RoboDK station: kr10 0621 Cube.rdk

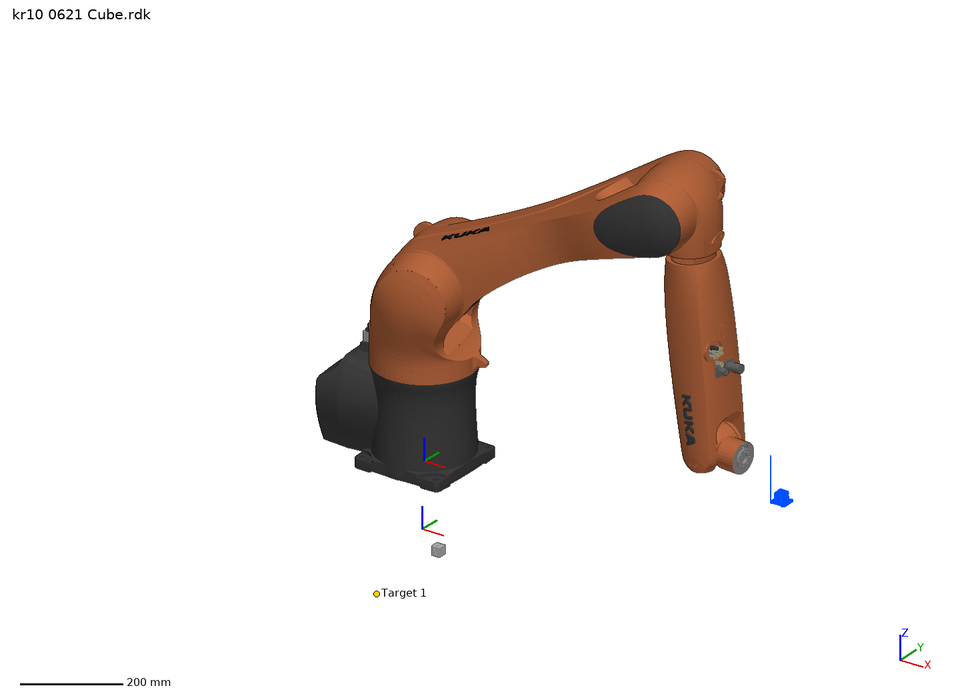
[picture v0: the station drawn from its stored meshes, robots at their saved joint values, targets as dots, program paths as lines]
Station kr10 0621 Cube. Poses are relative to the parent item; angles as X-Y-Z fixed-axis rotations.
  - frame KUKA KR 10 R1100 sixx Base at (0, 61.06, 0) mm
    - robot KUKA KR 10 R1100 sixx: 6 axes, payload 10 kg, reach 1101 mm, repeatability 0.03 mm, weight 54 kg
        modified DH rows (alpha deg, a mm, theta deg, d mm): 0, 0, 0, 400; -90, 25, 0, 0; 0, 560, -90, 0; -90, 35, 0, 515; 90, 0, 0, 0; -90, 0, 180, 80
        joint limits [-170, -190, -120, -185, -120, -350] to [170, 45, 156, 185, 120, 350]; home [0, -90, 90, 0, 0, 0]; saved at [-11.735, -27.383, 111.789, -15.728, -83.751, 50.742]
      - tool Tool 1, TCP at (31.57, 57.94, 75.73) mm, rotated rx -3.9 ry -0.86 rz 49.23 deg
    - frame Reference Rhino at (253.71, -369.34, 72) mm
      - object xyzCalibration_cube at (20, 0, -50) mm, size 20 x 20 x 20 mm, geometry from xyzCalibration_cube.stl
    - target Target 1 (Cartesian target) at (334.3, -640.64, 62.66) mm, rotated rx 170.43 ry 75.23 rz 170.98 deg; joints [61.963, -1.992, 26.262, -87.249, 55.611, -203.218] of KUKA KR 10 R1100 sixx
  - object box at (500, 500, 500) mm, size 250 x 250 x 250 mm, geometry from box.sld
  - machining project Print3D settings: C:/Users/Svassigh/Downloads/XYZ_20mm_Calibration_Cube/CFFFP_xyzCalibration_cube.gcode | rotZ(0) | rotX(0)*rotY(0)
  - Python program Extruder (listed below)
  - program Print3D (25115 instructions, listed below)
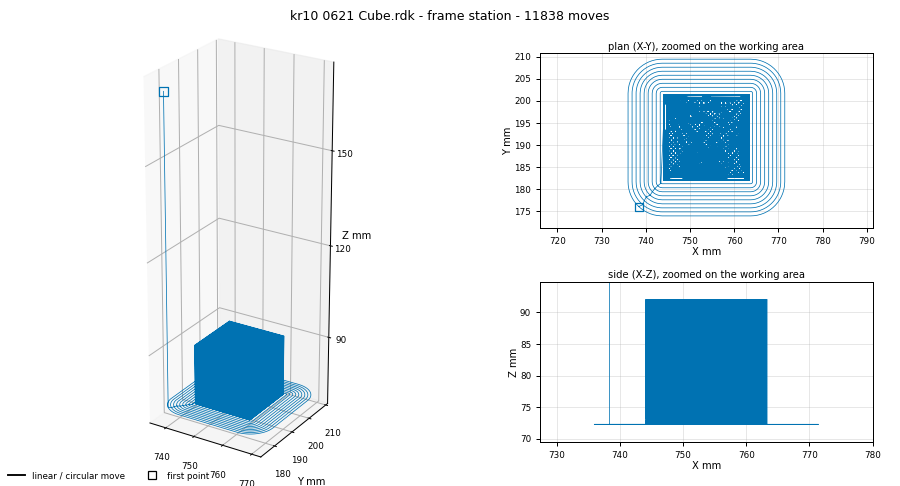
[picture p0: tool path of kr10 0621 Cube.rdk in frame station, 11838 of 11838 moves have a stored position in this frame; points joined in program order, loops and branches not executed]

--- Python program Extruder ---
# -*- coding: utf-8 -*-
"""
Created on Fri May 24 11:08:35 2019

@author: Rez
"""

import telnetlib
import sys

tn = telnetlib.Telnet('192.168.1.112', 23)
tn.read_until(b"Smoothie command shell")
str1 = str(sys.argv[1])
str2 = "G1 E" + str1 + " F200\n"
str3 = str2.encode('utf-8')
tn.write(str3)
tn.read_until(b"ok")
tn.write(b"exit")
tn.close
exit

--- program Print3D (robot KUKA KR 10 R1100 sixx) ---
  Smooth(10)
  Set Ref.: Reference Rhino
  Set Tool: Tool 1
  Show Tool 1
  Call M_RunCode(104)
  Call SetRPM(200.0)
  Call M_RunCode(105)
  Call M_RunCode(109)
  Call SetRPM(200.0)
  Call M_RunCode(82)
  Call Extruder(0.000)
  Set speed (3.3 mm/s)
  Call Extruder(3.000)
  Set speed (1000.0 mm/s)
  MoveJ 1 to (484.69, 484.38, 100.3) mm, rotated rx 0 ry 90 rz 0 deg; joints [-10.841, -37.414, 117.418, -14.997, -79.475, 51.803]
  MoveL 2 to (484.69, 484.38, 100.3) mm, rotated rx 0 ry 90 rz 0 deg; joints [-10.841, -37.414, 117.418, -14.997, -79.475, 51.803]
  MoveL 3 to (484.69, 484.38, 0.3) mm, rotated rx 0 ry 90 rz 0 deg; joints [-10.841, -26.609, 112.931, -14.783, -85.581, 50.166]
  MoveL 4 to (484.69, 484.38, 0.3) mm, rotated rx 0 ry 90 rz 0 deg; joints [-10.841, -26.609, 112.931, -14.783, -85.581, 50.166]
  Call Extruder(0.000)
  Call M_RunCode(83)
  Set speed (30.0 mm/s)
  Call Extruder(-0.400)
  MoveL 5 to (484.69, 484.38, 0.3) mm, rotated rx 0 ry 90 rz 0 deg; joints [-10.841, -26.609, 112.931, -14.783, -85.581, 50.166]
  Call M_RunCode(107)
  Set speed (60.0 mm/s)
  MoveL 6 to (484.69, 484.38, 0.3) mm, rotated rx 0 ry 90 rz 0 deg; joints [-10.841, -26.609, 112.931, -14.783, -85.581, 50.166]
  Set speed (30.0 mm/s)
  Call Extruder(0.400)
  MoveL 7 to (484.69, 484.38, 0.3) mm, rotated rx 0 ry 90 rz 0 deg; joints [-10.841, -26.609, 112.931, -14.783, -85.581, 50.166]
  Set speed (15.0 mm/s)
  Call Extruder(0.089)
  MoveL 8 to (485.29, 483.87, 0.3) mm, rotated rx 0 ry 90 rz 0 deg; joints [-10.782, -26.602, 112.872, -14.725, -85.53, 50.176]
  Call Extruder(0.089)
  MoveL 9 to (485.93, 483.42, 0.3) mm, rotated rx 0 ry 90 rz 0 deg; joints [-10.728, -26.594, 112.806, -14.672, -85.473, 50.187]
  Call Extruder(0.089)
  MoveL 10 to (486.62, 483.04, 0.3) mm, rotated rx 0 ry 90 rz 0 deg; joints [-10.68, -26.586, 112.734, -14.625, -85.411, 50.2]
  Call Extruder(0.089)
  MoveL 11 to (487.35, 482.74, 0.3) mm, rotated rx 0 ry 90 rz 0 deg; joints [-10.638, -26.576, 112.656, -14.584, -85.344, 50.215]
  Call Extruder(0.089)
  MoveL 12 to (488.1, 482.5, 0.3) mm, rotated rx 0 ry 90 rz 0 deg; joints [-10.603, -26.566, 112.573, -14.551, -85.272, 50.231]
  Call Extruder(0.089)
  MoveL 13 to (488.87, 482.35, 0.3) mm, rotated rx 0 ry 90 rz 0 deg; joints [-10.575, -26.555, 112.485, -14.524, -85.198, 50.248]
  Call Extruder(0.129)
  MoveL 14 to (490, 482.27, 0.3) mm, rotated rx 0 ry 90 rz 0 deg; joints [-10.547, -26.538, 112.354, -14.499, -85.086, 50.275]
  Call Extruder(2.270)
  MoveL 15 to (510, 482.26, 0.3) mm, rotated rx 0 ry 90 rz 0 deg; joints [-10.208, -26.205, 109.972, -14.21, -83.093, 50.756]
  Call Extruder(0.089)
  MoveL 16 to (510.79, 482.31, 0.3) mm, rotated rx 0 ry 90 rz 0 deg; joints [-10.198, -26.19, 109.876, -14.203, -83.015, 50.775]
  Call Extruder(0.089)
  MoveL 17 to (511.56, 482.42, 0.3) mm, rotated rx 0 ry 90 rz 0 deg; joints [-10.196, -26.176, 109.78, -14.204, -82.936, 50.794]
  Call Extruder(0.089)
  MoveL 18 to (512.32, 482.62, 0.3) mm, rotated rx 0 ry 90 rz 0 deg; joints [-10.202, -26.161, 109.684, -14.212, -82.857, 50.815]
  Call Extruder(0.089)
  MoveL 19 to (513.06, 482.9, 0.3) mm, rotated rx 0 ry 90 rz 0 deg; joints [-10.215, -26.146, 109.589, -14.227, -82.78, 50.836]
  MoveL 20 to (513.77, 483.24, 0.3) mm, rotated rx 0 ry 90 rz 0 deg; joints [-10.235, -26.131, 109.496, -14.25, -82.705, 50.858]
  Call Extruder(0.089)
  MoveL 21 to (514.43, 483.66, 0.3) mm, rotated rx 0 ry 90 rz 0 deg; joints [-10.262, -26.117, 109.406, -14.279, -82.632, 50.88]
  Call Extruder(0.089)
  MoveL 22 to (515.05, 484.14, 0.3) mm, rotated rx 0 ry 90 rz 0 deg; joints [-10.295, -26.103, 109.32, -14.315, -82.563, 50.902]
  Call Extruder(0.089)
  MoveL 23 to (515.62, 484.69, 0.3) mm, rotated rx 0 ry 90 rz 0 deg; joints [-10.335, -26.09, 109.24, -14.358, -82.499, 50.923]
  Call Extruder(0.089)
  MoveL 24 to (516.13, 485.29, 0.3) mm, rotated rx 0 ry 90 rz 0 deg; joints [-10.381, -26.078, 109.164, -14.406, -82.439, 50.944]
  Call Extruder(0.089)
  MoveL 25 to (516.58, 485.93, 0.3) mm, rotated rx 0 ry 90 rz 0 deg; joints [-10.431, -26.067, 109.096, -14.459, -82.385, 50.965]
  Call Extruder(0.089)
  MoveL 26 to (516.96, 486.62, 0.3) mm, rotated rx 0 ry 90 rz 0 deg; joints [-10.487, -26.057, 109.034, -14.517, -82.337, 50.984]
  Call Extruder(0.089)
  MoveL 27 to (517.27, 487.35, 0.3) mm, rotated rx 0 ry 90 rz 0 deg; joints [-10.547, -26.049, 108.981, -14.579, -82.295, 51.003]
  Call Extruder(0.089)
  MoveL 28 to (517.5, 488.1, 0.3) mm, rotated rx 0 ry 90 rz 0 deg; joints [-10.611, -26.041, 108.936, -14.645, -82.261, 51.02]
  Call Extruder(0.089)
  MoveL 29 to (517.65, 488.87, 0.3) mm, rotated rx 0 ry 90 rz 0 deg; joints [-10.678, -26.035, 108.899, -14.713, -82.233, 51.036]
  Call Extruder(0.129)
  MoveL 30 to (517.73, 490, 0.3) mm, rotated rx 0 ry 90 rz 0 deg; joints [-10.778, -26.029, 108.863, -14.815, -82.207, 51.056]
  Call Extruder(2.270)
  MoveL 31 to (517.74, 510, 0.3) mm, rotated rx 0 ry 90 rz 0 deg; joints [-12.561, -25.946, 108.362, -16.631, -81.868, 51.393]
  Call Extruder(0.089)
  MoveL 32 to (517.7, 510.79, 0.3) mm, rotated rx 0 ry 90 rz 0 deg; joints [-12.632, -25.943, 108.346, -16.702, -81.857, 51.406]
  Call Extruder(0.089)
  MoveL 33 to (517.58, 511.56, 0.3) mm, rotated rx 0 ry 90 rz 0 deg; joints [-12.703, -25.942, 108.339, -16.774, -81.855, 51.416]
  Call Extruder(0.089)
  MoveL 34 to (517.38, 512.32, 0.3) mm, rotated rx 0 ry 90 rz 0 deg; joints [-12.774, -25.942, 108.342, -16.846, -81.86, 51.425]
  Call Extruder(0.089)
  MoveL 35 to (517.1, 513.06, 0.3) mm, rotated rx 0 ry 90 rz 0 deg; joints [-12.845, -25.944, 108.355, -16.917, -81.873, 51.431]
  MoveL 36 to (516.76, 513.77, 0.3) mm, rotated rx 0 ry 90 rz 0 deg; joints [-12.915, -25.948, 108.378, -16.986, -81.894, 51.434]
  Call Extruder(0.089)
  MoveL 37 to (516.34, 514.43, 0.3) mm, rotated rx 0 ry 90 rz 0 deg; joints [-12.982, -25.954, 108.41, -17.053, -81.921, 51.435]
  Call Extruder(0.089)
  MoveL 38 to (515.86, 515.05, 0.3) mm, rotated rx 0 ry 90 rz 0 deg; joints [-13.047, -25.961, 108.451, -17.117, -81.957, 51.433]
  Call Extruder(0.089)
  MoveL 39 to (515.31, 515.62, 0.3) mm, rotated rx 0 ry 90 rz 0 deg; joints [-13.108, -25.969, 108.5, -17.178, -81.998, 51.428]
  Call Extruder(0.089)
  MoveL 40 to (514.71, 516.13, 0.3) mm, rotated rx 0 ry 90 rz 0 deg; joints [-13.166, -25.979, 108.558, -17.234, -82.047, 51.421]
  Call Extruder(0.089)
  MoveL 41 to (514.07, 516.58, 0.3) mm, rotated rx 0 ry 90 rz 0 deg; joints [-13.219, -25.99, 108.624, -17.285, -82.101, 51.411]
  Call Extruder(0.089)
  MoveL 42 to (513.38, 516.96, 0.3) mm, rotated rx 0 ry 90 rz 0 deg; joints [-13.267, -26.002, 108.696, -17.331, -82.16, 51.399]
  Call Extruder(0.089)
  MoveL 43 to (512.65, 517.27, 0.3) mm, rotated rx 0 ry 90 rz 0 deg; joints [-13.309, -26.015, 108.774, -17.371, -82.224, 51.385]
  Call Extruder(0.089)
  MoveL 44 to (511.9, 517.5, 0.3) mm, rotated rx 0 ry 90 rz 0 deg; joints [-13.346, -26.028, 108.858, -17.405, -82.292, 51.368]
  Call Extruder(0.089)
  MoveL 45 to (511.13, 517.65, 0.3) mm, rotated rx 0 ry 90 rz 0 deg; joints [-13.376, -26.043, 108.946, -17.432, -82.364, 51.349]
  Call Extruder(0.129)
  MoveL 46 to (510, 517.74, 0.3) mm, rotated rx 0 ry 90 rz 0 deg; joints [-13.407, -26.065, 109.08, -17.46, -82.471, 51.319]
  Call Extruder(2.270)
  MoveL 47 to (490, 517.74, 0.3) mm, rotated rx 0 ry 90 rz 0 deg; joints [-13.846, -26.42, 111.452, -17.83, -84.407, 50.748]
  Call Extruder(0.089)
  MoveL 48 to (489.22, 517.7, 0.3) mm, rotated rx 0 ry 90 rz 0 deg; joints [-13.86, -26.432, 111.545, -17.842, -84.484, 50.724]
  Call Extruder(0.089)
  MoveL 49 to (488.44, 517.58, 0.3) mm, rotated rx 0 ry 90 rz 0 deg; joints [-13.867, -26.445, 111.64, -17.846, -84.562, 50.699]
  Call Extruder(0.089)
  MoveL 50 to (487.68, 517.38, 0.3) mm, rotated rx 0 ry 90 rz 0 deg; joints [-13.866, -26.458, 111.734, -17.843, -84.641, 50.674]
  Call Extruder(0.089)
  MoveL 51 to (486.94, 517.1, 0.3) mm, rotated rx 0 ry 90 rz 0 deg; joints [-13.857, -26.47, 111.828, -17.832, -84.718, 50.648]
  MoveL 52 to (486.23, 516.76, 0.3) mm, rotated rx 0 ry 90 rz 0 deg; joints [-13.841, -26.483, 111.921, -17.814, -84.794, 50.622]
  Call Extruder(0.089)
  MoveL 53 to (485.57, 516.34, 0.3) mm, rotated rx 0 ry 90 rz 0 deg; joints [-13.818, -26.494, 112.011, -17.788, -84.868, 50.597]
  Call Extruder(0.089)
  MoveL 54 to (484.95, 515.86, 0.3) mm, rotated rx 0 ry 90 rz 0 deg; joints [-13.787, -26.506, 112.097, -17.755, -84.938, 50.571]
  Call Extruder(0.089)
  MoveL 55 to (484.38, 515.31, 0.3) mm, rotated rx 0 ry 90 rz 0 deg; joints [-13.75, -26.516, 112.179, -17.716, -85.005, 50.547]
  Call Extruder(0.089)
  MoveL 56 to (483.87, 514.71, 0.3) mm, rotated rx 0 ry 90 rz 0 deg; joints [-13.706, -26.526, 112.255, -17.67, -85.068, 50.523]
  Call Extruder(0.089)
  MoveL 57 to (483.42, 514.07, 0.3) mm, rotated rx 0 ry 90 rz 0 deg; joints [-13.656, -26.535, 112.326, -17.618, -85.125, 50.501]
  Call Extruder(0.089)
  MoveL 58 to (483.04, 513.38, 0.3) mm, rotated rx 0 ry 90 rz 0 deg; joints [-13.6, -26.543, 112.389, -17.561, -85.177, 50.48]
  Call Extruder(0.089)
  MoveL 59 to (482.73, 512.65, 0.3) mm, rotated rx 0 ry 90 rz 0 deg; joints [-13.539, -26.55, 112.445, -17.499, -85.223, 50.461]
  Call Extruder(0.089)
  MoveL 60 to (482.5, 511.9, 0.3) mm, rotated rx 0 ry 90 rz 0 deg; joints [-13.475, -26.556, 112.493, -17.433, -85.261, 50.444]
  Call Extruder(0.089)
  MoveL 61 to (482.35, 511.13, 0.3) mm, rotated rx 0 ry 90 rz 0 deg; joints [-13.406, -26.561, 112.533, -17.364, -85.293, 50.429]
  Call Extruder(0.129)
  MoveL 62 to (482.26, 510, 0.3) mm, rotated rx 0 ry 90 rz 0 deg; joints [-13.302, -26.566, 112.574, -17.258, -85.325, 50.412]
  Call Extruder(2.270)
  MoveL 63 to (482.27, 490, 0.3) mm, rotated rx 0 ry 90 rz 0 deg; joints [-11.419, -26.628, 113.085, -15.36, -85.721, 50.166]
  Call Extruder(0.089)
  MoveL 64 to (482.3, 489.21, 0.3) mm, rotated rx 0 ry 90 rz 0 deg; joints [-11.344, -26.629, 113.099, -15.285, -85.732, 50.158]
  Call Extruder(0.089)
  MoveL 65 to (482.42, 488.44, 0.3) mm, rotated rx 0 ry 90 rz 0 deg; joints [-11.268, -26.63, 113.103, -15.208, -85.734, 50.153]
  Call Extruder(0.089)
  MoveL 66 to (482.62, 487.68, 0.3) mm, rotated rx 0 ry 90 rz 0 deg; joints [-11.192, -26.629, 113.097, -15.132, -85.728, 50.15]
  Call Extruder(0.089)
  MoveL 67 to (482.9, 486.94, 0.3) mm, rotated rx 0 ry 90 rz 0 deg; joints [-11.117, -26.627, 113.082, -15.057, -85.714, 50.148]
  MoveL 68 to (483.24, 486.23, 0.3) mm, rotated rx 0 ry 90 rz 0 deg; joints [-11.044, -26.624, 113.058, -14.984, -85.692, 50.15]
  Call Extruder(0.089)
  MoveL 69 to (483.66, 485.57, 0.3) mm, rotated rx 0 ry 90 rz 0 deg; joints [-10.973, -26.62, 113.024, -14.914, -85.663, 50.153]
  Call Extruder(0.089)
  MoveL 70 to (484.14, 484.95, 0.3) mm, rotated rx 0 ry 90 rz 0 deg; joints [-10.905, -26.615, 112.982, -14.847, -85.625, 50.159]
  Call Extruder(0.089)
  MoveL 71 to (484.69, 484.38, 0.3) mm, rotated rx 0 ry 90 rz 0 deg; joints [-10.841, -26.609, 112.931, -14.783, -85.581, 50.166]
  Set speed (60.0 mm/s)
  MoveL 72 to (485.58, 484.8, 0.3) mm, rotated rx 0 ry 90 rz 0 deg; joints [-10.865, -26.596, 112.817, -14.809, -85.484, 50.193]
  Set speed (15.0 mm/s)
  Call Extruder(0.084)
  MoveL 73 to (486.17, 484.35, 0.3) mm, rotated rx 0 ry 90 rz 0 deg; joints [-10.812, -26.589, 112.758, -14.757, -85.433, 50.203]
  Call Extruder(0.084)
  MoveL 74 to (486.8, 483.97, 0.3) mm, rotated rx 0 ry 90 rz 0 deg; joints [-10.765, -26.58, 112.692, -14.711, -85.377, 50.215]
  Call Extruder(0.084)
  MoveL 75 to (487.47, 483.66, 0.3) mm, rotated rx 0 ry 90 rz 0 deg; joints [-10.723, -26.572, 112.621, -14.671, -85.315, 50.228]
  MoveL 76 to (488.17, 483.43, 0.3) mm, rotated rx 0 ry 90 rz 0 deg; joints [-10.688, -26.562, 112.544, -14.637, -85.249, 50.243]
  Call Extruder(0.084)
  MoveL 77 to (488.89, 483.27, 0.3) mm, rotated rx 0 ry 90 rz 0 deg; joints [-10.661, -26.552, 112.462, -14.611, -85.18, 50.259]
  Call Extruder(0.084)
  MoveL 78 to (489.63, 483.19, 0.3) mm, rotated rx 0 ry 90 rz 0 deg; joints [-10.64, -26.541, 112.378, -14.592, -85.108, 50.276]
  Call Extruder(0.042)
  MoveL 79 to (490, 483.18, 0.3) mm, rotated rx 0 ry 90 rz 0 deg; joints [-10.632, -26.536, 112.334, -14.585, -85.071, 50.285]
  Call Extruder(2.270)
  MoveL 80 to (510, 483.18, 0.3) mm, rotated rx 0 ry 90 rz 0 deg; joints [-10.291, -26.202, 109.952, -14.294, -83.079, 50.769]
  Call Extruder(0.084)
  MoveL 81 to (510.74, 483.22, 0.3) mm, rotated rx 0 ry 90 rz 0 deg; joints [-10.282, -26.188, 109.862, -14.288, -83.006, 50.786]
  Call Extruder(0.084)
  MoveL 82 to (511.47, 483.33, 0.3) mm, rotated rx 0 ry 90 rz 0 deg; joints [-10.281, -26.174, 109.772, -14.289, -82.932, 50.805]
  Call Extruder(0.084)
  MoveL 83 to (512.18, 483.53, 0.3) mm, rotated rx 0 ry 90 rz 0 deg; joints [-10.287, -26.16, 109.681, -14.298, -82.858, 50.825]
  Call Extruder(0.084)
  MoveL 84 to (512.86, 483.81, 0.3) mm, rotated rx 0 ry 90 rz 0 deg; joints [-10.301, -26.146, 109.593, -14.314, -82.786, 50.845]
  Call Extruder(0.084)
  MoveL 85 to (513.52, 484.15, 0.3) mm, rotated rx 0 ry 90 rz 0 deg; joints [-10.321, -26.133, 109.506, -14.337, -82.716, 50.866]
  Call Extruder(0.084)
  MoveL 86 to (514.13, 484.56, 0.3) mm, rotated rx 0 ry 90 rz 0 deg; joints [-10.348, -26.12, 109.423, -14.366, -82.649, 50.886]
  Call Extruder(0.084)
  MoveL 87 to (514.69, 485.04, 0.3) mm, rotated rx 0 ry 90 rz 0 deg; joints [-10.382, -26.107, 109.344, -14.403, -82.585, 50.907]
  Call Extruder(0.084)
  MoveL 88 to (515.2, 485.58, 0.3) mm, rotated rx 0 ry 90 rz 0 deg; joints [-10.422, -26.095, 109.271, -14.445, -82.527, 50.927]
  Call Extruder(0.084)
  MoveL 89 to (515.65, 486.17, 0.3) mm, rotated rx 0 ry 90 rz 0 deg; joints [-10.468, -26.085, 109.204, -14.493, -82.474, 50.946]
  Call Extruder(0.084)
  MoveL 90 to (516.03, 486.8, 0.3) mm, rotated rx 0 ry 90 rz 0 deg; joints [-10.519, -26.075, 109.143, -14.546, -82.426, 50.965]
  Call Extruder(0.084)
  MoveL 91 to (516.34, 487.47, 0.3) mm, rotated rx 0 ry 90 rz 0 deg; joints [-10.574, -26.066, 109.09, -14.603, -82.385, 50.983]
  MoveL 92 to (516.57, 488.17, 0.3) mm, rotated rx 0 ry 90 rz 0 deg; joints [-10.633, -26.059, 109.046, -14.664, -82.351, 50.999]
  Call Extruder(0.084)
  MoveL 93 to (516.73, 488.89, 0.3) mm, rotated rx 0 ry 90 rz 0 deg; joints [-10.695, -26.053, 109.01, -14.727, -82.324, 51.014]
  Call Extruder(0.084)
  MoveL 94 to (516.81, 489.63, 0.3) mm, rotated rx 0 ry 90 rz 0 deg; joints [-10.76, -26.049, 108.983, -14.793, -82.304, 51.028]
  Call Extruder(0.042)
  MoveL 95 to (516.83, 490, 0.3) mm, rotated rx 0 ry 90 rz 0 deg; joints [-10.793, -26.047, 108.974, -14.827, -82.297, 51.034]
  Call Extruder(2.270)
  MoveL 96 to (516.83, 510, 0.3) mm, rotated rx 0 ry 90 rz 0 deg; joints [-12.579, -25.964, 108.472, -16.645, -81.956, 51.369]
  Call Extruder(0.084)
  MoveL 97 to (516.79, 510.74, 0.3) mm, rotated rx 0 ry 90 rz 0 deg; joints [-12.646, -25.962, 108.457, -16.712, -81.947, 51.381]
  Call Extruder(0.084)
  MoveL 98 to (516.67, 511.47, 0.3) mm, rotated rx 0 ry 90 rz 0 deg; joints [-12.713, -25.961, 108.452, -16.78, -81.945, 51.39]
  Call Extruder(0.084)
  MoveL 99 to (516.47, 512.18, 0.3) mm, rotated rx 0 ry 90 rz 0 deg; joints [-12.78, -25.962, 108.456, -16.848, -81.951, 51.398]
  Call Extruder(0.084)
  MoveL 100 to (516.19, 512.86, 0.3) mm, rotated rx 0 ry 90 rz 0 deg; joints [-12.846, -25.964, 108.47, -16.914, -81.965, 51.403]
  Call Extruder(0.084)
  MoveL 101 to (515.85, 513.52, 0.3) mm, rotated rx 0 ry 90 rz 0 deg; joints [-12.911, -25.968, 108.494, -16.979, -81.986, 51.405]
  Call Extruder(0.084)
  MoveL 102 to (515.44, 514.13, 0.3) mm, rotated rx 0 ry 90 rz 0 deg; joints [-12.974, -25.973, 108.527, -17.041, -82.015, 51.405]
  Call Extruder(0.084)
  MoveL 103 to (514.96, 514.69, 0.3) mm, rotated rx 0 ry 90 rz 0 deg; joints [-13.033, -25.98, 108.569, -17.1, -82.05, 51.402]
  Call Extruder(0.084)
  MoveL 104 to (514.42, 515.2, 0.3) mm, rotated rx 0 ry 90 rz 0 deg; joints [-13.089, -25.989, 108.62, -17.154, -82.093, 51.396]
  Call Extruder(0.084)
  MoveL 105 to (513.83, 515.65, 0.3) mm, rotated rx 0 ry 90 rz 0 deg; joints [-13.141, -25.999, 108.678, -17.205, -82.141, 51.388]
  Call Extruder(0.084)
  MoveL 106 to (513.2, 516.03, 0.3) mm, rotated rx 0 ry 90 rz 0 deg; joints [-13.188, -26.009, 108.744, -17.25, -82.195, 51.378]
  Call Extruder(0.084)
  MoveL 107 to (512.53, 516.34, 0.3) mm, rotated rx 0 ry 90 rz 0 deg; joints [-13.23, -26.021, 108.815, -17.289, -82.254, 51.365]
  MoveL 108 to (511.83, 516.58, 0.3) mm, rotated rx 0 ry 90 rz 0 deg; joints [-13.265, -26.034, 108.893, -17.323, -82.317, 51.35]
  Call Extruder(0.084)
  MoveL 109 to (511.11, 516.73, 0.3) mm, rotated rx 0 ry 90 rz 0 deg; joints [-13.295, -26.048, 108.975, -17.349, -82.384, 51.332]
  Call Extruder(0.084)
  MoveL 110 to (510.37, 516.82, 0.3) mm, rotated rx 0 ry 90 rz 0 deg; joints [-13.317, -26.062, 109.061, -17.369, -82.453, 51.313]
  Call Extruder(0.042)
  MoveL 111 to (510, 516.83, 0.3) mm, rotated rx 0 ry 90 rz 0 deg; joints [-13.326, -26.069, 109.106, -17.377, -82.489, 51.303]
  Call Extruder(2.270)
  MoveL 112 to (490, 516.82, 0.3) mm, rotated rx 0 ry 90 rz 0 deg; joints [-13.762, -26.423, 111.478, -17.746, -84.427, 50.734]
  Call Extruder(0.084)
  MoveL 113 to (489.26, 516.79, 0.3) mm, rotated rx 0 ry 90 rz 0 deg; joints [-13.775, -26.435, 111.566, -17.756, -84.499, 50.712]
  Call Extruder(0.084)
  MoveL 114 to (488.53, 516.67, 0.3) mm, rotated rx 0 ry 90 rz 0 deg; joints [-13.781, -26.447, 111.654, -17.76, -84.572, 50.689]
  Call Extruder(0.084)
  MoveL 115 to (487.82, 516.47, 0.3) mm, rotated rx 0 ry 90 rz 0 deg; joints [-13.778, -26.459, 111.744, -17.755, -84.646, 50.665]
  Call Extruder(0.084)
  MoveL 116 to (487.14, 516.2, 0.3) mm, rotated rx 0 ry 90 rz 0 deg; joints [-13.769, -26.471, 111.832, -17.743, -84.718, 50.641]
  Call Extruder(0.084)
  MoveL 117 to (486.48, 515.85, 0.3) mm, rotated rx 0 ry 90 rz 0 deg; joints [-13.752, -26.482, 111.918, -17.724, -84.789, 50.616]
  Call Extruder(0.084)
  MoveL 118 to (485.87, 515.44, 0.3) mm, rotated rx 0 ry 90 rz 0 deg; joints [-13.727, -26.493, 112.001, -17.698, -84.858, 50.592]
  Call Extruder(0.084)
  MoveL 119 to (485.31, 514.96, 0.3) mm, rotated rx 0 ry 90 rz 0 deg; joints [-13.696, -26.503, 112.08, -17.664, -84.923, 50.569]
  Call Extruder(0.084)
  MoveL 120 to (484.8, 514.42, 0.3) mm, rotated rx 0 ry 90 rz 0 deg; joints [-13.657, -26.513, 112.155, -17.624, -84.984, 50.546]
  Call Extruder(0.084)
  MoveL 121 to (484.35, 513.83, 0.3) mm, rotated rx 0 ry 90 rz 0 deg; joints [-13.613, -26.522, 112.224, -17.578, -85.04, 50.525]
  Call Extruder(0.084)
  MoveL 122 to (483.97, 513.2, 0.3) mm, rotated rx 0 ry 90 rz 0 deg; joints [-13.563, -26.53, 112.286, -17.526, -85.09, 50.505]
  Call Extruder(0.084)
  MoveL 123 to (483.66, 512.53, 0.3) mm, rotated rx 0 ry 90 rz 0 deg; joints [-13.507, -26.537, 112.341, -17.469, -85.135, 50.487]
  MoveL 124 to (483.43, 511.83, 0.3) mm, rotated rx 0 ry 90 rz 0 deg; joints [-13.447, -26.543, 112.388, -17.408, -85.173, 50.47]
  Call Extruder(0.084)
  MoveL 125 to (483.27, 511.11, 0.3) mm, rotated rx 0 ry 90 rz 0 deg; joints [-13.384, -26.548, 112.427, -17.343, -85.204, 50.456]
  Call Extruder(0.084)
  MoveL 126 to (483.19, 510.37, 0.3) mm, rotated rx 0 ry 90 rz 0 deg; joints [-13.317, -26.551, 112.456, -17.276, -85.227, 50.443]
  Call Extruder(0.042)
  MoveL 127 to (483.17, 510, 0.3) mm, rotated rx 0 ry 90 rz 0 deg; joints [-13.282, -26.553, 112.468, -17.241, -85.236, 50.438]
  Call Extruder(2.270)
  MoveL 128 to (483.17, 490, 0.3) mm, rotated rx 0 ry 90 rz 0 deg; joints [-11.402, -26.615, 112.979, -15.345, -85.631, 50.19]
  Call Extruder(0.084)
  MoveL 129 to (483.22, 489.26, 0.3) mm, rotated rx 0 ry 90 rz 0 deg; joints [-11.331, -26.617, 112.991, -15.274, -85.64, 50.183]
  Call Extruder(0.084)
  MoveL 130 to (483.33, 488.53, 0.3) mm, rotated rx 0 ry 90 rz 0 deg; joints [-11.26, -26.617, 112.994, -15.202, -85.642, 50.177]
  Call Extruder(0.084)
  MoveL 131 to (483.53, 487.82, 0.3) mm, rotated rx 0 ry 90 rz 0 deg; joints [-11.189, -26.616, 112.988, -15.131, -85.635, 50.175]
  Call Extruder(0.084)
  MoveL 132 to (483.81, 487.14, 0.3) mm, rotated rx 0 ry 90 rz 0 deg; joints [-11.119, -26.614, 112.972, -15.061, -85.62, 50.174]
  Call Extruder(0.084)
  MoveL 133 to (484.15, 486.48, 0.3) mm, rotated rx 0 ry 90 rz 0 deg; joints [-11.051, -26.611, 112.946, -14.993, -85.597, 50.176]
  Call Extruder(0.084)
  MoveL 134 to (484.57, 485.87, 0.3) mm, rotated rx 0 ry 90 rz 0 deg; joints [-10.985, -26.607, 112.912, -14.928, -85.567, 50.179]
  Call Extruder(0.084)
  MoveL 135 to (485.04, 485.31, 0.3) mm, rotated rx 0 ry 90 rz 0 deg; joints [-10.923, -26.602, 112.868, -14.866, -85.529, 50.185]
  Call Extruder(0.084)
  MoveL 136 to (485.58, 484.8, 0.3) mm, rotated rx 0 ry 90 rz 0 deg; joints [-10.865, -26.596, 112.817, -14.809, -85.484, 50.193]
  Set speed (60.0 mm/s)
  MoveL 137 to (485.94, 485.7, 0.3) mm, rotated rx 0 ry 90 rz 0 deg; joints [-10.943, -26.588, 112.754, -14.889, -85.433, 50.212]
  Set speed (15.0 mm/s)
  Call Extruder(0.078)
  MoveL 138 to (486.47, 485.26, 0.3) mm, rotated rx 0 ry 90 rz 0 deg; joints [-10.892, -26.582, 112.703, -14.838, -85.388, 50.221]
  Call Extruder(0.078)
  MoveL 139 to (487.04, 484.88, 0.3) mm, rotated rx 0 ry 90 rz 0 deg; joints [-10.846, -26.575, 112.644, -14.793, -85.337, 50.231]
  Call Extruder(0.078)
  MoveL 140 to (487.65, 484.57, 0.3) mm, rotated rx 0 ry 90 rz 0 deg; joints [-10.806, -26.566, 112.579, -14.754, -85.281, 50.243]
  Call Extruder(0.078)
  MoveL 141 to (488.3, 484.33, 0.3) mm, rotated rx 0 ry 90 rz 0 deg; joints [-10.772, -26.558, 112.508, -14.721, -85.221, 50.256]
  Call Extruder(0.078)
  MoveL 142 to (488.97, 484.18, 0.3) mm, rotated rx 0 ry 90 rz 0 deg; joints [-10.745, -26.548, 112.433, -14.696, -85.157, 50.271]
  MoveL 143 to (489.65, 484.1, 0.3) mm, rotated rx 0 ry 90 rz 0 deg; joints [-10.725, -26.538, 112.354, -14.678, -85.09, 50.287]
  Call Extruder(0.039)
  MoveL 144 to (490, 484.08, 0.3) mm, rotated rx 0 ry 90 rz 0 deg; joints [-10.718, -26.533, 112.314, -14.671, -85.055, 50.296]
  Call Extruder(2.270)
  MoveL 145 to (510, 484.09, 0.3) mm, rotated rx 0 ry 90 rz 0 deg; joints [-10.373, -26.199, 109.932, -14.378, -83.065, 50.782]
  Call Extruder(0.078)
  MoveL 146 to (510.69, 484.12, 0.3) mm, rotated rx 0 ry 90 rz 0 deg; joints [-10.366, -26.186, 109.848, -14.373, -82.997, 50.798]
  Call Extruder(0.078)
  MoveL 147 to (511.36, 484.24, 0.3) mm, rotated rx 0 ry 90 rz 0 deg; joints [-10.365, -26.173, 109.764, -14.374, -82.928, 50.816]
  Call Extruder(0.078)
  MoveL 148 to (512.02, 484.44, 0.3) mm, rotated rx 0 ry 90 rz 0 deg; joints [-10.372, -26.16, 109.68, -14.383, -82.859, 50.835]
  Call Extruder(0.078)
  MoveL 149 to (512.65, 484.71, 0.3) mm, rotated rx 0 ry 90 rz 0 deg; joints [-10.386, -26.147, 109.598, -14.4, -82.792, 50.854]
  Call Extruder(0.078)
  MoveL 150 to (513.25, 485.06, 0.3) mm, rotated rx 0 ry 90 rz 0 deg; joints [-10.408, -26.135, 109.518, -14.423, -82.728, 50.873]
  Call Extruder(0.078)
  MoveL 151 to (513.8, 485.47, 0.3) mm, rotated rx 0 ry 90 rz 0 deg; joints [-10.436, -26.123, 109.443, -14.454, -82.667, 50.892]
  Call Extruder(0.078)
  MoveL 152 to (514.3, 485.94, 0.3) mm, rotated rx 0 ry 90 rz 0 deg; joints [-10.47, -26.111, 109.372, -14.49, -82.61, 50.911]
  Call Extruder(0.078)
  MoveL 153 to (514.74, 486.47, 0.3) mm, rotated rx 0 ry 90 rz 0 deg; joints [-10.51, -26.101, 109.306, -14.533, -82.558, 50.929]
  Call Extruder(0.078)
  MoveL 154 to (515.12, 487.04, 0.3) mm, rotated rx 0 ry 90 rz 0 deg; joints [-10.556, -26.092, 109.248, -14.58, -82.512, 50.947]
  Call Extruder(0.078)
  MoveL 155 to (515.43, 487.65, 0.3) mm, rotated rx 0 ry 90 rz 0 deg; joints [-10.606, -26.083, 109.196, -14.632, -82.472, 50.964]
  Call Extruder(0.078)
  MoveL 156 to (515.67, 488.3, 0.3) mm, rotated rx 0 ry 90 rz 0 deg; joints [-10.66, -26.076, 109.153, -14.688, -82.438, 50.98]
  Call Extruder(0.078)
  MoveL 157 to (515.83, 488.97, 0.3) mm, rotated rx 0 ry 90 rz 0 deg; joints [-10.718, -26.071, 109.119, -14.747, -82.412, 50.994]
  MoveL 158 to (515.91, 489.65, 0.3) mm, rotated rx 0 ry 90 rz 0 deg; joints [-10.778, -26.067, 109.093, -14.808, -82.393, 51.006]
  Call Extruder(0.039)
  MoveL 159 to (515.91, 490, 0.3) mm, rotated rx 0 ry 90 rz 0 deg; joints [-10.809, -26.065, 109.084, -14.84, -82.387, 51.012]
  Call Extruder(2.270)
  MoveL 160 to (515.91, 510, 0.3) mm, rotated rx 0 ry 90 rz 0 deg; joints [-12.597, -25.983, 108.582, -16.659, -82.045, 51.344]
  Call Extruder(0.078)
  MoveL 161 to (515.88, 510.69, 0.3) mm, rotated rx 0 ry 90 rz 0 deg; joints [-12.659, -25.98, 108.569, -16.722, -82.036, 51.355]
  Call Extruder(0.078)
  MoveL 162 to (515.76, 511.36, 0.3) mm, rotated rx 0 ry 90 rz 0 deg; joints [-12.722, -25.98, 108.565, -16.785, -82.035, 51.364]
  Call Extruder(0.078)
  MoveL 163 to (515.56, 512.02, 0.3) mm, rotated rx 0 ry 90 rz 0 deg; joints [-12.784, -25.981, 108.57, -16.848, -82.042, 51.371]
  Call Extruder(0.078)
  MoveL 164 to (515.29, 512.65, 0.3) mm, rotated rx 0 ry 90 rz 0 deg; joints [-12.846, -25.983, 108.586, -16.91, -82.057, 51.374]
  Call Extruder(0.078)
  MoveL 165 to (514.94, 513.25, 0.3) mm, rotated rx 0 ry 90 rz 0 deg; joints [-12.906, -25.987, 108.611, -16.969, -82.079, 51.376]
  Call Extruder(0.078)
  MoveL 166 to (514.53, 513.8, 0.3) mm, rotated rx 0 ry 90 rz 0 deg; joints [-12.963, -25.993, 108.645, -17.026, -82.108, 51.374]
  Call Extruder(0.078)
  MoveL 167 to (514.06, 514.3, 0.3) mm, rotated rx 0 ry 90 rz 0 deg; joints [-13.017, -26, 108.688, -17.079, -82.145, 51.37]
  Call Extruder(0.078)
  MoveL 168 to (513.53, 514.74, 0.3) mm, rotated rx 0 ry 90 rz 0 deg; joints [-13.067, -26.009, 108.739, -17.128, -82.187, 51.364]
  Call Extruder(0.078)
  MoveL 169 to (512.96, 515.12, 0.3) mm, rotated rx 0 ry 90 rz 0 deg; joints [-13.113, -26.019, 108.798, -17.172, -82.236, 51.355]
  Call Extruder(0.078)
  MoveL 170 to (512.35, 515.43, 0.3) mm, rotated rx 0 ry 90 rz 0 deg; joints [-13.153, -26.029, 108.863, -17.21, -82.289, 51.343]
  Call Extruder(0.078)
  MoveL 171 to (511.7, 515.67, 0.3) mm, rotated rx 0 ry 90 rz 0 deg; joints [-13.187, -26.041, 108.934, -17.243, -82.347, 51.33]
  Call Extruder(0.078)
  MoveL 172 to (511.03, 515.83, 0.3) mm, rotated rx 0 ry 90 rz 0 deg; joints [-13.215, -26.053, 109.01, -17.268, -82.409, 51.314]
  MoveL 173 to (510.35, 515.9, 0.3) mm, rotated rx 0 ry 90 rz 0 deg; joints [-13.237, -26.066, 109.09, -17.287, -82.474, 51.297]
  Call Extruder(0.039)
  MoveL 174 to (510, 515.91, 0.3) mm, rotated rx 0 ry 90 rz 0 deg; joints [-13.245, -26.073, 109.131, -17.294, -82.507, 51.287]
  Call Extruder(2.270)
  MoveL 175 to (490, 515.92, 0.3) mm, rotated rx 0 ry 90 rz 0 deg; joints [-13.679, -26.427, 111.504, -17.661, -84.446, 50.72]
  Call Extruder(0.078)
  MoveL 176 to (489.31, 515.88, 0.3) mm, rotated rx 0 ry 90 rz 0 deg; joints [-13.69, -26.438, 111.586, -17.671, -84.514, 50.699]
  Call Extruder(0.078)
  MoveL 177 to (488.64, 515.76, 0.3) mm, rotated rx 0 ry 90 rz 0 deg; joints [-13.694, -26.449, 111.669, -17.673, -84.582, 50.678]
  Call Extruder(0.078)
  MoveL 178 to (487.98, 515.56, 0.3) mm, rotated rx 0 ry 90 rz 0 deg; joints [-13.691, -26.46, 111.751, -17.667, -84.65, 50.656]
  Call Extruder(0.078)
  MoveL 179 to (487.35, 515.29, 0.3) mm, rotated rx 0 ry 90 rz 0 deg; joints [-13.68, -26.471, 111.833, -17.654, -84.717, 50.633]
  Call Extruder(0.078)
  MoveL 180 to (486.75, 514.94, 0.3) mm, rotated rx 0 ry 90 rz 0 deg; joints [-13.662, -26.481, 111.912, -17.634, -84.782, 50.611]
  Call Extruder(0.078)
  MoveL 181 to (486.2, 514.53, 0.3) mm, rotated rx 0 ry 90 rz 0 deg; joints [-13.636, -26.491, 111.988, -17.607, -84.845, 50.589]
  Call Extruder(0.078)
  MoveL 182 to (485.7, 514.06, 0.3) mm, rotated rx 0 ry 90 rz 0 deg; joints [-13.604, -26.501, 112.06, -17.572, -84.904, 50.568]
  Call Extruder(0.078)
  MoveL 183 to (485.26, 513.53, 0.3) mm, rotated rx 0 ry 90 rz 0 deg; joints [-13.565, -26.509, 112.127, -17.532, -84.958, 50.547]
  Call Extruder(0.078)
  MoveL 184 to (484.88, 512.96, 0.3) mm, rotated rx 0 ry 90 rz 0 deg; joints [-13.52, -26.517, 112.187, -17.485, -85.007, 50.528]
  Call Extruder(0.078)
  MoveL 185 to (484.57, 512.35, 0.3) mm, rotated rx 0 ry 90 rz 0 deg; joints [-13.47, -26.524, 112.24, -17.434, -85.05, 50.51]
  Call Extruder(0.078)
  MoveL 186 to (484.33, 511.7, 0.3) mm, rotated rx 0 ry 90 rz 0 deg; joints [-13.415, -26.53, 112.286, -17.378, -85.087, 50.495]
  Call Extruder(0.078)
  MoveL 187 to (484.18, 511.03, 0.3) mm, rotated rx 0 ry 90 rz 0 deg; joints [-13.356, -26.534, 112.323, -17.318, -85.116, 50.481]
  MoveL 188 to (484.09, 510.35, 0.3) mm, rotated rx 0 ry 90 rz 0 deg; joints [-13.294, -26.538, 112.351, -17.255, -85.139, 50.469]
  Call Extruder(0.039)
  MoveL 189 to (484.09, 510, 0.3) mm, rotated rx 0 ry 90 rz 0 deg; joints [-13.262, -26.539, 112.362, -17.223, -85.147, 50.464]
  Call Extruder(2.270)
  MoveL 190 to (484.09, 490, 0.3) mm, rotated rx 0 ry 90 rz 0 deg; joints [-11.385, -26.602, 112.872, -15.329, -85.54, 50.214]
  Call Extruder(0.078)
  MoveL 191 to (484.12, 489.31, 0.3) mm, rotated rx 0 ry 90 rz 0 deg; joints [-11.319, -26.604, 112.884, -15.263, -85.549, 50.207]
  Call Extruder(0.078)
  MoveL 192 to (484.24, 488.64, 0.3) mm, rotated rx 0 ry 90 rz 0 deg; joints [-11.253, -26.604, 112.886, -15.197, -85.549, 50.202]
  Call Extruder(0.078)
  MoveL 193 to (484.44, 487.98, 0.3) mm, rotated rx 0 ry 90 rz 0 deg; joints [-11.187, -26.603, 112.878, -15.131, -85.541, 50.2]
  Call Extruder(0.078)
  MoveL 194 to (484.71, 487.35, 0.3) mm, rotated rx 0 ry 90 rz 0 deg; joints [-11.122, -26.601, 112.86, -15.066, -85.526, 50.2]
  Call Extruder(0.078)
  MoveL 195 to (485.06, 486.75, 0.3) mm, rotated rx 0 ry 90 rz 0 deg; joints [-11.059, -26.598, 112.834, -15.004, -85.502, 50.202]
  Call Extruder(0.078)
  MoveL 196 to (485.47, 486.2, 0.3) mm, rotated rx 0 ry 90 rz 0 deg; joints [-10.999, -26.593, 112.798, -14.944, -85.471, 50.206]
  Call Extruder(0.078)
  MoveL 197 to (485.94, 485.7, 0.3) mm, rotated rx 0 ry 90 rz 0 deg; joints [-10.943, -26.588, 112.754, -14.889, -85.433, 50.212]
  Set speed (60.0 mm/s)
  MoveL 198 to (486.37, 486.56, 0.3) mm, rotated rx 0 ry 90 rz 0 deg; joints [-11.017, -26.58, 112.685, -14.964, -85.375, 50.233]
  Set speed (15.0 mm/s)
  Call Extruder(0.072)
  MoveL 199 to (486.83, 486.13, 0.3) mm, rotated rx 0 ry 90 rz 0 deg; joints [-10.967, -26.574, 112.64, -14.915, -85.336, 50.24]
  Call Extruder(0.072)
  MoveL 200 to (487.34, 485.76, 0.3) mm, rotated rx 0 ry 90 rz 0 deg; joints [-10.923, -26.568, 112.588, -14.872, -85.291, 50.249]
  Call Extruder(0.072)
  MoveL 201 to (487.9, 485.46, 0.3) mm, rotated rx 0 ry 90 rz 0 deg; joints [-10.885, -26.56, 112.53, -14.834, -85.241, 50.259]
  Call Extruder(0.072)
  MoveL 202 to (488.49, 485.23, 0.3) mm, rotated rx 0 ry 90 rz 0 deg; joints [-10.853, -26.552, 112.466, -14.803, -85.186, 50.272]
  MoveL 203 to (489.1, 485.08, 0.3) mm, rotated rx 0 ry 90 rz 0 deg; joints [-10.827, -26.544, 112.397, -14.779, -85.128, 50.285]
  Call Extruder(0.102)
  MoveL 204 to (490, 484.99, 0.3) mm, rotated rx 0 ry 90 rz 0 deg; joints [-10.804, -26.531, 112.293, -14.757, -85.04, 50.307]
  Call Extruder(2.270)
  MoveL 205 to (510, 485, 0.3) mm, rotated rx 0 ry 90 rz 0 deg; joints [-10.456, -26.196, 109.912, -14.462, -83.051, 50.795]
  Call Extruder(0.072)
  MoveL 206 to (510.63, 485.04, 0.3) mm, rotated rx 0 ry 90 rz 0 deg; joints [-10.449, -26.184, 109.835, -14.457, -82.988, 50.81]
  Call Extruder(0.072)
  MoveL 207 to (511.25, 485.15, 0.3) mm, rotated rx 0 ry 90 rz 0 deg; joints [-10.45, -26.172, 109.757, -14.46, -82.924, 50.827]
  Call Extruder(0.072)
  MoveL 208 to (511.85, 485.35, 0.3) mm, rotated rx 0 ry 90 rz 0 deg; joints [-10.458, -26.16, 109.68, -14.47, -82.862, 50.844]
  Call Extruder(0.072)
  MoveL 209 to (512.42, 485.62, 0.3) mm, rotated rx 0 ry 90 rz 0 deg; joints [-10.473, -26.148, 109.605, -14.487, -82.801, 50.862]
  Call Extruder(0.072)
  MoveL 210 to (512.96, 485.96, 0.3) mm, rotated rx 0 ry 90 rz 0 deg; joints [-10.495, -26.137, 109.533, -14.511, -82.743, 50.879]
  Call Extruder(0.072)
  MoveL 211 to (513.44, 486.37, 0.3) mm, rotated rx 0 ry 90 rz 0 deg; joints [-10.523, -26.126, 109.466, -14.541, -82.689, 50.897]
  Call Extruder(0.072)
  MoveL 212 to (513.87, 486.83, 0.3) mm, rotated rx 0 ry 90 rz 0 deg; joints [-10.558, -26.117, 109.403, -14.578, -82.639, 50.914]
  Call Extruder(0.072)
  MoveL 213 to (514.24, 487.35, 0.3) mm, rotated rx 0 ry 90 rz 0 deg; joints [-10.598, -26.108, 109.347, -14.62, -82.594, 50.931]
  Call Extruder(0.072)
  MoveL 214 to (514.54, 487.9, 0.3) mm, rotated rx 0 ry 90 rz 0 deg; joints [-10.643, -26.1, 109.298, -14.667, -82.556, 50.947]
  Call Extruder(0.072)
  MoveL 215 to (514.77, 488.49, 0.3) mm, rotated rx 0 ry 90 rz 0 deg; joints [-10.693, -26.093, 109.257, -14.718, -82.524, 50.961]
  MoveL 216 to (514.92, 489.11, 0.3) mm, rotated rx 0 ry 90 rz 0 deg; joints [-10.745, -26.088, 109.225, -14.772, -82.499, 50.974]
  Call Extruder(0.102)
  MoveL 217 to (515, 490, 0.3) mm, rotated rx 0 ry 90 rz 0 deg; joints [-10.825, -26.083, 109.194, -14.853, -82.477, 50.99]
  Call Extruder(2.270)
  MoveL 218 to (515.01, 510, 0.3) mm, rotated rx 0 ry 90 rz 0 deg; joints [-12.616, -26.001, 108.692, -16.674, -82.133, 51.32]
  Call Extruder(0.072)
  MoveL 219 to (514.97, 510.63, 0.3) mm, rotated rx 0 ry 90 rz 0 deg; joints [-12.672, -25.999, 108.68, -16.732, -82.125, 51.33]
  Call Extruder(0.072)
  MoveL 220 to (514.85, 511.25, 0.3) mm, rotated rx 0 ry 90 rz 0 deg; joints [-12.73, -25.999, 108.678, -16.79, -82.125, 51.338]
  Call Extruder(0.072)
  MoveL 221 to (514.65, 511.85, 0.3) mm, rotated rx 0 ry 90 rz 0 deg; joints [-12.787, -26, 108.685, -16.848, -82.133, 51.343]
  Call Extruder(0.072)
  MoveL 222 to (514.38, 512.42, 0.3) mm, rotated rx 0 ry 90 rz 0 deg; joints [-12.844, -26.003, 108.702, -16.904, -82.149, 51.346]
  Call Extruder(0.072)
  MoveL 223 to (514.04, 512.96, 0.3) mm, rotated rx 0 ry 90 rz 0 deg; joints [-12.898, -26.007, 108.728, -16.958, -82.172, 51.346]
  Call Extruder(0.072)
  MoveL 224 to (513.63, 513.44, 0.3) mm, rotated rx 0 ry 90 rz 0 deg; joints [-12.949, -26.013, 108.764, -17.008, -82.202, 51.344]
  Call Extruder(0.072)
  MoveL 225 to (513.17, 513.87, 0.3) mm, rotated rx 0 ry 90 rz 0 deg; joints [-12.997, -26.02, 108.808, -17.055, -82.239, 51.338]
  Call Extruder(0.072)
  MoveL 226 to (512.65, 514.24, 0.3) mm, rotated rx 0 ry 90 rz 0 deg; joints [-13.041, -26.029, 108.859, -17.097, -82.282, 51.331]
  Call Extruder(0.072)
  MoveL 227 to (512.1, 514.54, 0.3) mm, rotated rx 0 ry 90 rz 0 deg; joints [-13.079, -26.038, 108.918, -17.134, -82.33, 51.321]
  Call Extruder(0.072)
  MoveL 228 to (511.51, 514.77, 0.3) mm, rotated rx 0 ry 90 rz 0 deg; joints [-13.112, -26.049, 108.982, -17.165, -82.383, 51.309]
  MoveL 229 to (510.9, 514.92, 0.3) mm, rotated rx 0 ry 90 rz 0 deg; joints [-13.138, -26.06, 109.052, -17.189, -82.439, 51.295]
  Call Extruder(0.102)
  MoveL 230 to (510, 515, 0.3) mm, rotated rx 0 ry 90 rz 0 deg; joints [-13.164, -26.077, 109.157, -17.212, -82.525, 51.271]
  Call Extruder(2.270)
  MoveL 231 to (490, 515.01, 0.3) mm, rotated rx 0 ry 90 rz 0 deg; joints [-13.595, -26.43, 111.53, -17.576, -84.465, 50.706]
  Call Extruder(0.072)
  MoveL 232 to (489.37, 514.96, 0.3) mm, rotated rx 0 ry 90 rz 0 deg; joints [-13.605, -26.441, 111.605, -17.585, -84.527, 50.687]
  Call Extruder(0.072)
  MoveL 233 to (488.75, 514.85, 0.3) mm, rotated rx 0 ry 90 rz 0 deg; joints [-13.608, -26.451, 111.681, -17.586, -84.59, 50.668]
  Call Extruder(0.072)
  MoveL 234 to (488.15, 514.65, 0.3) mm, rotated rx 0 ry 90 rz 0 deg; joints [-13.603, -26.461, 111.757, -17.579, -84.653, 50.647]
  Call Extruder(0.072)
  MoveL 235 to (487.58, 514.38, 0.3) mm, rotated rx 0 ry 90 rz 0 deg; joints [-13.591, -26.471, 111.832, -17.565, -84.714, 50.627]
  Call Extruder(0.072)
  MoveL 236 to (487.04, 514.04, 0.3) mm, rotated rx 0 ry 90 rz 0 deg; joints [-13.572, -26.48, 111.904, -17.544, -84.773, 50.606]
  Call Extruder(0.072)
  MoveL 237 to (486.56, 513.63, 0.3) mm, rotated rx 0 ry 90 rz 0 deg; joints [-13.545, -26.489, 111.972, -17.515, -84.829, 50.586]
  Call Extruder(0.072)
  MoveL 238 to (486.13, 513.17, 0.3) mm, rotated rx 0 ry 90 rz 0 deg; joints [-13.512, -26.498, 112.035, -17.48, -84.881, 50.567]
  Call Extruder(0.072)
  MoveL 239 to (485.76, 512.65, 0.3) mm, rotated rx 0 ry 90 rz 0 deg; joints [-13.472, -26.505, 112.093, -17.44, -84.928, 50.549]
  Call Extruder(0.072)
  MoveL 240 to (485.46, 512.1, 0.3) mm, rotated rx 0 ry 90 rz 0 deg; joints [-13.427, -26.512, 112.144, -17.393, -84.969, 50.533]
  Call Extruder(0.072)
  MoveL 241 to (485.23, 511.51, 0.3) mm, rotated rx 0 ry 90 rz 0 deg; joints [-13.377, -26.517, 112.187, -17.342, -85.004, 50.518]
  MoveL 242 to (485.08, 510.89, 0.3) mm, rotated rx 0 ry 90 rz 0 deg; joints [-13.324, -26.522, 112.221, -17.288, -85.031, 50.505]
  Call Extruder(0.102)
  MoveL 243 to (485, 510, 0.3) mm, rotated rx 0 ry 90 rz 0 deg; joints [-13.242, -26.526, 112.256, -17.205, -85.058, 50.49]
  Call Extruder(2.270)
  MoveL 244 to (484.99, 490, 0.3) mm, rotated rx 0 ry 90 rz 0 deg; joints [-11.367, -26.589, 112.766, -15.314, -85.45, 50.237]
  Call Extruder(0.072)
  MoveL 245 to (485.04, 489.37, 0.3) mm, rotated rx 0 ry 90 rz 0 deg; joints [-11.307, -26.591, 112.776, -15.253, -85.457, 50.231]
  Call Extruder(0.072)
  MoveL 246 to (485.15, 488.75, 0.3) mm, rotated rx 0 ry 90 rz 0 deg; joints [-11.246, -26.591, 112.776, -15.192, -85.456, 50.227]
  Call Extruder(0.072)
  MoveL 247 to (485.35, 488.15, 0.3) mm, rotated rx 0 ry 90 rz 0 deg; joints [-11.186, -26.59, 112.767, -15.132, -85.448, 50.225]
  Call Extruder(0.072)
  MoveL 248 to (485.62, 487.57, 0.3) mm, rotated rx 0 ry 90 rz 0 deg; joints [-11.127, -26.587, 112.749, -15.073, -85.431, 50.226]
  Call Extruder(0.072)
  MoveL 249 to (485.96, 487.04, 0.3) mm, rotated rx 0 ry 90 rz 0 deg; joints [-11.07, -26.584, 112.721, -15.017, -85.407, 50.228]
  Call Extruder(0.072)
  MoveL 250 to (486.37, 486.56, 0.3) mm, rotated rx 0 ry 90 rz 0 deg; joints [-11.017, -26.58, 112.685, -14.964, -85.375, 50.233]
  Set speed (60.0 mm/s)
  MoveL 251 to (487.26, 486.95, 0.3) mm, rotated rx 0 ry 90 rz 0 deg; joints [-11.038, -26.566, 112.571, -14.987, -85.278, 50.26]
  Set speed (15.0 mm/s)
  Call Extruder(0.065)
  MoveL 252 to (487.71, 486.6, 0.3) mm, rotated rx 0 ry 90 rz 0 deg; joints [-10.996, -26.56, 112.526, -14.946, -85.24, 50.268]
  MoveL 253 to (488.21, 486.32, 0.3) mm, rotated rx 0 ry 90 rz 0 deg; joints [-10.96, -26.553, 112.474, -14.911, -85.195, 50.277]
  Call Extruder(0.065)
  MoveL 254 to (488.74, 486.1, 0.3) mm, rotated rx 0 ry 90 rz 0 deg; joints [-10.93, -26.546, 112.416, -14.882, -85.146, 50.288]
  Call Extruder(0.065)
  MoveL 255 to (489.3, 485.97, 0.3) mm, rotated rx 0 ry 90 rz 0 deg; joints [-10.908, -26.538, 112.354, -14.861, -85.093, 50.3]
  Call Extruder(0.080)
  MoveL 256 to (490, 485.91, 0.3) mm, rotated rx 0 ry 90 rz 0 deg; joints [-10.889, -26.528, 112.273, -14.844, -85.024, 50.317]
  Call Extruder(2.270)
  MoveL 257 to (510, 485.91, 0.3) mm, rotated rx 0 ry 90 rz 0 deg; joints [-10.539, -26.193, 109.891, -14.546, -83.037, 50.808]
  Call Extruder(0.065)
  MoveL 258 to (510.57, 485.95, 0.3) mm, rotated rx 0 ry 90 rz 0 deg; joints [-10.533, -26.182, 109.822, -14.542, -82.979, 50.822]
  Call Extruder(0.065)
  MoveL 259 to (511.13, 486.06, 0.3) mm, rotated rx 0 ry 90 rz 0 deg; joints [-10.535, -26.171, 109.752, -14.545, -82.922, 50.837]
  Call Extruder(0.065)
  MoveL 260 to (511.67, 486.26, 0.3) mm, rotated rx 0 ry 90 rz 0 deg; joints [-10.543, -26.16, 109.682, -14.556, -82.866, 50.853]
  Call Extruder(0.065)
  MoveL 261 to (512.17, 486.53, 0.3) mm, rotated rx 0 ry 90 rz 0 deg; joints [-10.559, -26.15, 109.616, -14.574, -82.812, 50.869]
  Call Extruder(0.065)
  MoveL 262 to (512.63, 486.87, 0.3) mm, rotated rx 0 ry 90 rz 0 deg; joints [-10.582, -26.14, 109.552, -14.598, -82.761, 50.885]
  Call Extruder(0.065)
  MoveL 263 to (513.05, 487.26, 0.3) mm, rotated rx 0 ry 90 rz 0 deg; joints [-10.611, -26.131, 109.494, -14.629, -82.714, 50.901]
  Call Extruder(0.065)
  MoveL 264 to (513.4, 487.71, 0.3) mm, rotated rx 0 ry 90 rz 0 deg; joints [-10.646, -26.122, 109.441, -14.665, -82.672, 50.916]
  MoveL 265 to (513.68, 488.21, 0.3) mm, rotated rx 0 ry 90 rz 0 deg; joints [-10.686, -26.115, 109.395, -14.707, -82.636, 50.931]
  Call Extruder(0.065)
  MoveL 266 to (513.9, 488.74, 0.3) mm, rotated rx 0 ry 90 rz 0 deg; joints [-10.73, -26.109, 109.357, -14.753, -82.606, 50.944]
  Call Extruder(0.065)
  MoveL 267 to (514.03, 489.3, 0.3) mm, rotated rx 0 ry 90 rz 0 deg; joints [-10.778, -26.104, 109.328, -14.802, -82.584, 50.956]
  Call Extruder(0.080)
  MoveL 268 to (514.1, 490, 0.3) mm, rotated rx 0 ry 90 rz 0 deg; joints [-10.84, -26.101, 109.304, -14.865, -82.566, 50.968]
  Call Extruder(2.270)
  MoveL 269 to (514.09, 510, 0.3) mm, rotated rx 0 ry 90 rz 0 deg; joints [-12.634, -26.019, 108.802, -16.689, -82.221, 51.296]
  Call Extruder(0.065)
  MoveL 270 to (514.05, 510.57, 0.3) mm, rotated rx 0 ry 90 rz 0 deg; joints [-12.685, -26.017, 108.792, -16.741, -82.215, 51.305]
  Call Extruder(0.065)
  MoveL 271 to (513.94, 511.13, 0.3) mm, rotated rx 0 ry 90 rz 0 deg; joints [-12.738, -26.017, 108.791, -16.794, -82.216, 51.311]
  Call Extruder(0.065)
  MoveL 272 to (513.74, 511.67, 0.3) mm, rotated rx 0 ry 90 rz 0 deg; joints [-12.789, -26.019, 108.8, -16.846, -82.225, 51.315]
  Call Extruder(0.065)
  MoveL 273 to (513.47, 512.17, 0.3) mm, rotated rx 0 ry 90 rz 0 deg; joints [-12.84, -26.022, 108.818, -16.896, -82.242, 51.317]
  Call Extruder(0.065)
  MoveL 274 to (513.13, 512.63, 0.3) mm, rotated rx 0 ry 90 rz 0 deg; joints [-12.888, -26.026, 108.846, -16.943, -82.266, 51.316]
  Call Extruder(0.065)
  MoveL 275 to (512.74, 513.05, 0.3) mm, rotated rx 0 ry 90 rz 0 deg; joints [-12.932, -26.032, 108.883, -16.987, -82.297, 51.312]
  Call Extruder(0.065)
  MoveL 276 to (512.29, 513.4, 0.3) mm, rotated rx 0 ry 90 rz 0 deg; joints [-12.973, -26.04, 108.927, -17.027, -82.334, 51.306]
  MoveL 277 to (511.79, 513.68, 0.3) mm, rotated rx 0 ry 90 rz 0 deg; joints [-13.009, -26.048, 108.979, -17.061, -82.376, 51.297]
  Call Extruder(0.065)
  MoveL 278 to (511.26, 513.9, 0.3) mm, rotated rx 0 ry 90 rz 0 deg; joints [-13.039, -26.058, 109.037, -17.089, -82.424, 51.287]
  Call Extruder(0.065)
  MoveL 279 to (510.7, 514.03, 0.3) mm, rotated rx 0 ry 90 rz 0 deg; joints [-13.062, -26.068, 109.1, -17.111, -82.475, 51.274]
  Call Extruder(0.080)
  MoveL 280 to (510, 514.1, 0.3) mm, rotated rx 0 ry 90 rz 0 deg; joints [-13.082, -26.081, 109.183, -17.129, -82.542, 51.256]
  Call Extruder(2.270)
  MoveL 281 to (490, 514.1, 0.3) mm, rotated rx 0 ry 90 rz 0 deg; joints [-13.511, -26.434, 111.556, -17.492, -84.484, 50.693]
  Call Extruder(0.065)
  MoveL 282 to (489.43, 514.05, 0.3) mm, rotated rx 0 ry 90 rz 0 deg; joints [-13.52, -26.443, 111.624, -17.499, -84.541, 50.676]
  Call Extruder(0.065)
  MoveL 283 to (488.87, 513.94, 0.3) mm, rotated rx 0 ry 90 rz 0 deg; joints [-13.521, -26.452, 111.693, -17.499, -84.598, 50.658]
  Call Extruder(0.065)
  MoveL 284 to (488.33, 513.74, 0.3) mm, rotated rx 0 ry 90 rz 0 deg; joints [-13.515, -26.461, 111.761, -17.491, -84.654, 50.639]
  Call Extruder(0.065)
  MoveL 285 to (487.83, 513.47, 0.3) mm, rotated rx 0 ry 90 rz 0 deg; joints [-13.502, -26.47, 111.828, -17.475, -84.709, 50.621]
  Call Extruder(0.065)
  MoveL 286 to (487.37, 513.14, 0.3) mm, rotated rx 0 ry 90 rz 0 deg; joints [-13.481, -26.479, 111.892, -17.453, -84.761, 50.603]
  Call Extruder(0.065)
  MoveL 287 to (486.95, 512.74, 0.3) mm, rotated rx 0 ry 90 rz 0 deg; joints [-13.453, -26.486, 111.951, -17.424, -84.809, 50.585]
  Call Extruder(0.065)
  MoveL 288 to (486.6, 512.29, 0.3) mm, rotated rx 0 ry 90 rz 0 deg; joints [-13.419, -26.494, 112.005, -17.388, -84.853, 50.568]
  MoveL 289 to (486.32, 511.79, 0.3) mm, rotated rx 0 ry 90 rz 0 deg; joints [-13.379, -26.5, 112.052, -17.348, -84.891, 50.553]
  Call Extruder(0.065)
  MoveL 290 to (486.1, 511.26, 0.3) mm, rotated rx 0 ry 90 rz 0 deg; joints [-13.335, -26.505, 112.091, -17.302, -84.923, 50.54]
  Call Extruder(0.065)
  MoveL 291 to (485.97, 510.7, 0.3) mm, rotated rx 0 ry 90 rz 0 deg; joints [-13.286, -26.509, 112.123, -17.252, -84.948, 50.528]
  Call Extruder(0.080)
  MoveL 292 to (485.91, 510, 0.3) mm, rotated rx 0 ry 90 rz 0 deg; joints [-13.222, -26.512, 112.149, -17.188, -84.969, 50.516]
  Call Extruder(2.270)
  MoveL 293 to (485.91, 490, 0.3) mm, rotated rx 0 ry 90 rz 0 deg; joints [-11.35, -26.576, 112.659, -15.299, -85.359, 50.261]
  Call Extruder(0.065)
  MoveL 294 to (485.95, 489.43, 0.3) mm, rotated rx 0 ry 90 rz 0 deg; joints [-11.295, -26.578, 112.668, -15.244, -85.365, 50.255]
  Call Extruder(0.065)
  MoveL 295 to (486.06, 488.87, 0.3) mm, rotated rx 0 ry 90 rz 0 deg; joints [-11.241, -26.577, 112.667, -15.189, -85.364, 50.252]
  Call Extruder(0.065)
  MoveL 296 to (486.26, 488.33, 0.3) mm, rotated rx 0 ry 90 rz 0 deg; joints [-11.186, -26.576, 112.657, -15.134, -85.354, 50.251]
  Call Extruder(0.065)
  MoveL 297 to (486.53, 487.83, 0.3) mm, rotated rx 0 ry 90 rz 0 deg; joints [-11.134, -26.574, 112.637, -15.082, -85.336, 50.252]
  Call Extruder(0.065)
  MoveL 298 to (486.87, 487.37, 0.3) mm, rotated rx 0 ry 90 rz 0 deg; joints [-11.084, -26.57, 112.608, -15.032, -85.311, 50.255]
  Call Extruder(0.065)
  MoveL 299 to (487.26, 486.95, 0.3) mm, rotated rx 0 ry 90 rz 0 deg; joints [-11.038, -26.566, 112.571, -14.987, -85.278, 50.26]
  Set speed (60.0 mm/s)
  MoveL 300 to (487.76, 487.73, 0.3) mm, rotated rx 0 ry 90 rz 0 deg; joints [-11.102, -26.556, 112.494, -15.053, -85.215, 50.282]
  Set speed (15.0 mm/s)
  Call Extruder(0.057)
  MoveL 301 to (488.15, 487.41, 0.3) mm, rotated rx 0 ry 90 rz 0 deg; joints [-11.064, -26.551, 112.456, -15.016, -85.182, 50.288]
  MoveL 302 to (488.58, 487.15, 0.3) mm, rotated rx 0 ry 90 rz 0 deg; joints [-11.032, -26.546, 112.411, -14.984, -85.143, 50.296]
  Call Extruder(0.057)
  MoveL 303 to (489.05, 486.96, 0.3) mm, rotated rx 0 ry 90 rz 0 deg; joints [-11.005, -26.539, 112.36, -14.959, -85.1, 50.306]
  Call Extruder(0.057)
  MoveL 304 to (489.54, 486.85, 0.3) mm, rotated rx 0 ry 90 rz 0 deg; joints [-10.986, -26.532, 112.305, -14.94, -85.053, 50.317]
  Call Extruder(0.052)
  MoveL 305 to (490, 486.82, 0.3) mm, rotated rx 0 ry 90 rz 0 deg; joints [-10.974, -26.525, 112.252, -14.93, -85.008, 50.328]
  Call Extruder(2.270)
  MoveL 306 to (510, 486.82, 0.3) mm, rotated rx 0 ry 90 rz 0 deg; joints [-10.622, -26.19, 109.871, -14.63, -83.022, 50.821]
  Call Extruder(0.057)
  MoveL 307 to (510.5, 486.86, 0.3) mm, rotated rx 0 ry 90 rz 0 deg; joints [-10.617, -26.18, 109.809, -14.627, -82.972, 50.834]
  Call Extruder(0.057)
  MoveL 308 to (510.99, 486.97, 0.3) mm, rotated rx 0 ry 90 rz 0 deg; joints [-10.62, -26.171, 109.748, -14.631, -82.921, 50.847]
  Call Extruder(0.057)
  MoveL 309 to (511.46, 487.17, 0.3) mm, rotated rx 0 ry 90 rz 0 deg; joints [-10.629, -26.161, 109.687, -14.642, -82.872, 50.861]
  Call Extruder(0.057)
  MoveL 310 to (511.89, 487.43, 0.3) mm, rotated rx 0 ry 90 rz 0 deg; joints [-10.646, -26.152, 109.63, -14.661, -82.826, 50.876]
  Call Extruder(0.057)
  MoveL 311 to (512.27, 487.76, 0.3) mm, rotated rx 0 ry 90 rz 0 deg; joints [-10.669, -26.144, 109.576, -14.686, -82.783, 50.89]
  Call Extruder(0.057)
  MoveL 312 to (512.59, 488.15, 0.3) mm, rotated rx 0 ry 90 rz 0 deg; joints [-10.699, -26.136, 109.528, -14.717, -82.744, 50.903]
  MoveL 313 to (512.85, 488.58, 0.3) mm, rotated rx 0 ry 90 rz 0 deg; joints [-10.734, -26.13, 109.487, -14.753, -82.712, 50.916]
  Call Extruder(0.057)
  MoveL 314 to (513.04, 489.05, 0.3) mm, rotated rx 0 ry 90 rz 0 deg; joints [-10.773, -26.124, 109.453, -14.793, -82.686, 50.928]
  Call Extruder(0.057)
  MoveL 315 to (513.15, 489.54, 0.3) mm, rotated rx 0 ry 90 rz 0 deg; joints [-10.815, -26.121, 109.429, -14.837, -82.667, 50.938]
  Call Extruder(0.052)
  MoveL 316 to (513.18, 490, 0.3) mm, rotated rx 0 ry 90 rz 0 deg; joints [-10.856, -26.118, 109.414, -14.878, -82.656, 50.946]
  Call Extruder(2.270)
  MoveL 317 to (513.18, 510, 0.3) mm, rotated rx 0 ry 90 rz 0 deg; joints [-12.652, -26.037, 108.912, -16.704, -82.31, 51.271]
  Call Extruder(0.057)
  MoveL 318 to (513.15, 510.5, 0.3) mm, rotated rx 0 ry 90 rz 0 deg; joints [-12.698, -26.036, 108.903, -16.75, -82.305, 51.279]
  Call Extruder(0.057)
  MoveL 319 to (513.03, 510.99, 0.3) mm, rotated rx 0 ry 90 rz 0 deg; joints [-12.744, -26.036, 108.904, -16.796, -82.307, 51.284]
  Call Extruder(0.057)
  MoveL 320 to (512.83, 511.46, 0.3) mm, rotated rx 0 ry 90 rz 0 deg; joints [-12.789, -26.038, 108.915, -16.842, -82.317, 51.287]
  Call Extruder(0.057)
  MoveL 321 to (512.57, 511.89, 0.3) mm, rotated rx 0 ry 90 rz 0 deg; joints [-12.833, -26.041, 108.935, -16.885, -82.335, 51.287]
  Call Extruder(0.057)
  MoveL 322 to (512.24, 512.27, 0.3) mm, rotated rx 0 ry 90 rz 0 deg; joints [-12.873, -26.046, 108.964, -16.925, -82.36, 51.285]
  Call Extruder(0.057)
  MoveL 323 to (511.85, 512.59, 0.3) mm, rotated rx 0 ry 90 rz 0 deg; joints [-12.91, -26.052, 109.002, -16.961, -82.391, 51.28]
  MoveL 324 to (511.42, 512.85, 0.3) mm, rotated rx 0 ry 90 rz 0 deg; joints [-12.942, -26.059, 109.047, -16.992, -82.428, 51.273]
  Call Extruder(0.057)
  MoveL 325 to (510.95, 513.04, 0.3) mm, rotated rx 0 ry 90 rz 0 deg; joints [-12.969, -26.068, 109.098, -17.017, -82.47, 51.263]
  Call Extruder(0.057)
  MoveL 326 to (510.46, 513.15, 0.3) mm, rotated rx 0 ry 90 rz 0 deg; joints [-12.989, -26.077, 109.154, -17.035, -82.516, 51.252]
  Call Extruder(0.052)
  MoveL 327 to (510, 513.18, 0.3) mm, rotated rx 0 ry 90 rz 0 deg; joints [-13.001, -26.085, 109.208, -17.046, -82.559, 51.24]
  Call Extruder(2.270)
  MoveL 328 to (490, 513.19, 0.3) mm, rotated rx 0 ry 90 rz 0 deg; joints [-13.427, -26.437, 111.581, -17.407, -84.503, 50.679]
  Call Extruder(0.057)
  MoveL 329 to (489.5, 513.14, 0.3) mm, rotated rx 0 ry 90 rz 0 deg; joints [-13.435, -26.445, 111.642, -17.413, -84.553, 50.664]
  Call Extruder(0.057)
  MoveL 330 to (489.01, 513.03, 0.3) mm, rotated rx 0 ry 90 rz 0 deg; joints [-13.434, -26.454, 111.702, -17.411, -84.603, 50.648]
  Call Extruder(0.057)
  MoveL 331 to (488.54, 512.83, 0.3) mm, rotated rx 0 ry 90 rz 0 deg; joints [-13.427, -26.462, 111.762, -17.402, -84.653, 50.632]
  Call Extruder(0.057)
  MoveL 332 to (488.11, 512.57, 0.3) mm, rotated rx 0 ry 90 rz 0 deg; joints [-13.412, -26.469, 111.82, -17.385, -84.7, 50.616]
  Call Extruder(0.057)
  MoveL 333 to (487.73, 512.24, 0.3) mm, rotated rx 0 ry 90 rz 0 deg; joints [-13.39, -26.476, 111.874, -17.362, -84.744, 50.6]
  Call Extruder(0.057)
  MoveL 334 to (487.41, 511.85, 0.3) mm, rotated rx 0 ry 90 rz 0 deg; joints [-13.361, -26.483, 111.923, -17.332, -84.784, 50.585]
  MoveL 335 to (487.15, 511.42, 0.3) mm, rotated rx 0 ry 90 rz 0 deg; joints [-13.327, -26.488, 111.965, -17.296, -84.818, 50.572]
  Call Extruder(0.057)
  MoveL 336 to (486.96, 510.95, 0.3) mm, rotated rx 0 ry 90 rz 0 deg; joints [-13.287, -26.493, 112, -17.256, -84.846, 50.56]
  Call Extruder(0.057)
  MoveL 337 to (486.85, 510.46, 0.3) mm, rotated rx 0 ry 90 rz 0 deg; joints [-13.244, -26.496, 112.026, -17.212, -84.867, 50.55]
  Call Extruder(0.052)
  MoveL 338 to (486.81, 510, 0.3) mm, rotated rx 0 ry 90 rz 0 deg; joints [-13.202, -26.499, 112.043, -17.17, -84.88, 50.542]
  Call Extruder(2.270)
  MoveL 339 to (486.81, 490, 0.3) mm, rotated rx 0 ry 90 rz 0 deg; joints [-11.333, -26.563, 112.552, -15.283, -85.268, 50.285]
  Call Extruder(0.057)
  MoveL 340 to (486.86, 489.5, 0.3) mm, rotated rx 0 ry 90 rz 0 deg; joints [-11.285, -26.564, 112.56, -15.235, -85.274, 50.28]
  Call Extruder(0.057)
  MoveL 341 to (486.97, 489.01, 0.3) mm, rotated rx 0 ry 90 rz 0 deg; joints [-11.236, -26.564, 112.557, -15.187, -85.271, 50.277]
  Call Extruder(0.057)
  MoveL 342 to (487.17, 488.54, 0.3) mm, rotated rx 0 ry 90 rz 0 deg; joints [-11.189, -26.562, 112.545, -15.139, -85.26, 50.276]
  Call Extruder(0.057)
  MoveL 343 to (487.43, 488.11, 0.3) mm, rotated rx 0 ry 90 rz 0 deg; joints [-11.144, -26.56, 112.524, -15.094, -85.241, 50.278]
  Call Extruder(0.057)
  MoveL 344 to (487.76, 487.73, 0.3) mm, rotated rx 0 ry 90 rz 0 deg; joints [-11.102, -26.556, 112.494, -15.053, -85.215, 50.282]
  Set speed (60.0 mm/s)
  MoveL 345 to (488.34, 488.45, 0.3) mm, rotated rx 0 ry 90 rz 0 deg; joints [-11.159, -26.545, 112.41, -15.111, -85.145, 50.305]
  Set speed (15.0 mm/s)
  Call Extruder(0.048)
  MoveL 346 to (488.65, 488.17, 0.3) mm, rotated rx 0 ry 90 rz 0 deg; joints [-11.126, -26.542, 112.379, -15.079, -85.118, 50.31]
  Call Extruder(0.048)
  MoveL 347 to (489.02, 487.95, 0.3) mm, rotated rx 0 ry 90 rz 0 deg; joints [-11.099, -26.537, 112.341, -15.053, -85.086, 50.317]
  Call Extruder(0.048)
  MoveL 348 to (489.42, 487.8, 0.3) mm, rotated rx 0 ry 90 rz 0 deg; joints [-11.078, -26.531, 112.298, -15.032, -85.049, 50.325]
  Call Extruder(0.066)
  MoveL 349 to (490, 487.73, 0.3) mm, rotated rx 0 ry 90 rz 0 deg; joints [-11.06, -26.523, 112.231, -15.016, -84.992, 50.339]
  Call Extruder(2.270)
  MoveL 350 to (510, 487.73, 0.3) mm, rotated rx 0 ry 90 rz 0 deg; joints [-10.705, -26.186, 109.85, -14.714, -83.008, 50.834]
  Call Extruder(0.048)
  MoveL 351 to (510.42, 487.76, 0.3) mm, rotated rx 0 ry 90 rz 0 deg; joints [-10.701, -26.178, 109.798, -14.712, -82.965, 50.845]
  Call Extruder(0.048)
  MoveL 352 to (510.83, 487.88, 0.3) mm, rotated rx 0 ry 90 rz 0 deg; joints [-10.705, -26.17, 109.746, -14.717, -82.923, 50.857]
  Call Extruder(0.048)
  MoveL 353 to (511.21, 488.08, 0.3) mm, rotated rx 0 ry 90 rz 0 deg; joints [-10.716, -26.163, 109.696, -14.729, -82.882, 50.869]
  Call Extruder(0.048)
  MoveL 354 to (511.55, 488.34, 0.3) mm, rotated rx 0 ry 90 rz 0 deg; joints [-10.734, -26.155, 109.65, -14.748, -82.844, 50.881]
  Call Extruder(0.048)
  MoveL 355 to (511.83, 488.65, 0.3) mm, rotated rx 0 ry 90 rz 0 deg; joints [-10.758, -26.149, 109.608, -14.774, -82.811, 50.893]
  Call Extruder(0.048)
  MoveL 356 to (512.05, 489.02, 0.3) mm, rotated rx 0 ry 90 rz 0 deg; joints [-10.787, -26.143, 109.573, -14.804, -82.784, 50.904]
  Call Extruder(0.048)
  MoveL 357 to (512.2, 489.42, 0.3) mm, rotated rx 0 ry 90 rz 0 deg; joints [-10.821, -26.139, 109.546, -14.839, -82.763, 50.913]
  Call Extruder(0.066)
  MoveL 358 to (512.27, 490, 0.3) mm, rotated rx 0 ry 90 rz 0 deg; joints [-10.872, -26.136, 109.524, -14.891, -82.746, 50.924]
  Call Extruder(2.270)
  MoveL 359 to (512.27, 510, 0.3) mm, rotated rx 0 ry 90 rz 0 deg; joints [-12.67, -26.055, 109.022, -16.718, -82.398, 51.247]
  Call Extruder(0.048)
  MoveL 360 to (512.24, 510.42, 0.3) mm, rotated rx 0 ry 90 rz 0 deg; joints [-12.709, -26.054, 109.015, -16.758, -82.394, 51.253]
  Call Extruder(0.048)
  MoveL 361 to (512.12, 510.83, 0.3) mm, rotated rx 0 ry 90 rz 0 deg; joints [-12.748, -26.055, 109.018, -16.797, -82.398, 51.257]
  Call Extruder(0.048)
  MoveL 362 to (511.92, 511.21, 0.3) mm, rotated rx 0 ry 90 rz 0 deg; joints [-12.786, -26.057, 109.031, -16.835, -82.41, 51.258]
  Call Extruder(0.048)
  MoveL 363 to (511.66, 511.55, 0.3) mm, rotated rx 0 ry 90 rz 0 deg; joints [-12.821, -26.06, 109.053, -16.869, -82.429, 51.257]
  Call Extruder(0.048)
  MoveL 364 to (511.35, 511.83, 0.3) mm, rotated rx 0 ry 90 rz 0 deg; joints [-12.853, -26.065, 109.083, -16.9, -82.454, 51.253]
  Call Extruder(0.048)
  MoveL 365 to (510.98, 512.05, 0.3) mm, rotated rx 0 ry 90 rz 0 deg; joints [-12.88, -26.071, 109.121, -16.926, -82.486, 51.247]
  Call Extruder(0.048)
  MoveL 366 to (510.58, 512.2, 0.3) mm, rotated rx 0 ry 90 rz 0 deg; joints [-12.901, -26.078, 109.165, -16.947, -82.522, 51.239]
  Call Extruder(0.066)
  MoveL 367 to (510, 512.28, 0.3) mm, rotated rx 0 ry 90 rz 0 deg; joints [-12.92, -26.089, 109.233, -16.963, -82.577, 51.224]
  Call Extruder(2.270)
  MoveL 368 to (490, 512.28, 0.3) mm, rotated rx 0 ry 90 rz 0 deg; joints [-13.343, -26.441, 111.607, -17.322, -84.522, 50.666]
  Call Extruder(0.048)
  MoveL 369 to (489.58, 512.24, 0.3) mm, rotated rx 0 ry 90 rz 0 deg; joints [-13.349, -26.448, 111.658, -17.326, -84.564, 50.653]
  Call Extruder(0.048)
  MoveL 370 to (489.17, 512.12, 0.3) mm, rotated rx 0 ry 90 rz 0 deg; joints [-13.347, -26.454, 111.709, -17.323, -84.607, 50.64]
  Call Extruder(0.048)
  MoveL 371 to (488.79, 511.92, 0.3) mm, rotated rx 0 ry 90 rz 0 deg; joints [-13.338, -26.461, 111.759, -17.312, -84.648, 50.626]
  Call Extruder(0.048)
  MoveL 372 to (488.45, 511.66, 0.3) mm, rotated rx 0 ry 90 rz 0 deg; joints [-13.321, -26.467, 111.806, -17.295, -84.686, 50.613]
  Call Extruder(0.048)
  MoveL 373 to (488.17, 511.35, 0.3) mm, rotated rx 0 ry 90 rz 0 deg; joints [-13.298, -26.473, 111.848, -17.27, -84.72, 50.6]
  Call Extruder(0.048)
  MoveL 374 to (487.95, 510.98, 0.3) mm, rotated rx 0 ry 90 rz 0 deg; joints [-13.269, -26.478, 111.883, -17.24, -84.749, 50.588]
  Call Extruder(0.048)
  MoveL 375 to (487.8, 510.58, 0.3) mm, rotated rx 0 ry 90 rz 0 deg; joints [-13.235, -26.481, 111.912, -17.206, -84.772, 50.579]
  Call Extruder(0.066)
  MoveL 376 to (487.73, 510, 0.3) mm, rotated rx 0 ry 90 rz 0 deg; joints [-13.183, -26.485, 111.936, -17.153, -84.791, 50.568]
  Call Extruder(2.270)
  MoveL 377 to (487.73, 490, 0.3) mm, rotated rx 0 ry 90 rz 0 deg; joints [-11.316, -26.55, 112.446, -15.268, -85.178, 50.308]
  Call Extruder(0.048)
  MoveL 378 to (487.77, 489.58, 0.3) mm, rotated rx 0 ry 90 rz 0 deg; joints [-11.275, -26.551, 112.451, -15.227, -85.182, 50.304]
  Call Extruder(0.048)
  MoveL 379 to (487.88, 489.17, 0.3) mm, rotated rx 0 ry 90 rz 0 deg; joints [-11.234, -26.55, 112.447, -15.187, -85.177, 50.302]
  Call Extruder(0.048)
  MoveL 380 to (488.08, 488.79, 0.3) mm, rotated rx 0 ry 90 rz 0 deg; joints [-11.195, -26.548, 112.433, -15.147, -85.165, 50.303]
  Call Extruder(0.048)
  MoveL 381 to (488.34, 488.45, 0.3) mm, rotated rx 0 ry 90 rz 0 deg; joints [-11.159, -26.545, 112.41, -15.111, -85.145, 50.305]
  Set speed (60.0 mm/s)
  MoveL 382 to (488.98, 489.09, 0.3) mm, rotated rx 0 ry 90 rz 0 deg; joints [-11.207, -26.534, 112.319, -15.162, -85.069, 50.33]
  Set speed (15.0 mm/s)
  Call Extruder(0.037)
  MoveL 383 to (489.23, 488.88, 0.3) mm, rotated rx 0 ry 90 rz 0 deg; joints [-11.182, -26.531, 112.295, -15.137, -85.049, 50.333]
  Call Extruder(0.038)
  MoveL 384 to (489.52, 488.72, 0.3) mm, rotated rx 0 ry 90 rz 0 deg; joints [-11.162, -26.527, 112.265, -15.118, -85.022, 50.339]
  Call Extruder(0.055)
  MoveL 385 to (490, 488.64, 0.3) mm, rotated rx 0 ry 90 rz 0 deg; joints [-11.145, -26.52, 112.21, -15.102, -84.976, 50.35]
  Call Extruder(2.270)
  MoveL 386 to (510, 488.64, 0.3) mm, rotated rx 0 ry 90 rz 0 deg; joints [-10.788, -26.183, 109.83, -14.798, -82.993, 50.848]
  Call Extruder(0.037)
  MoveL 387 to (510.33, 488.68, 0.3) mm, rotated rx 0 ry 90 rz 0 deg; joints [-10.786, -26.177, 109.789, -14.797, -82.96, 50.856]
  Call Extruder(0.037)
  MoveL 388 to (510.64, 488.79, 0.3) mm, rotated rx 0 ry 90 rz 0 deg; joints [-10.791, -26.171, 109.749, -14.803, -82.928, 50.866]
  Call Extruder(0.037)
  MoveL 389 to (510.91, 488.98, 0.3) mm, rotated rx 0 ry 90 rz 0 deg; joints [-10.803, -26.165, 109.712, -14.817, -82.898, 50.875]
  Call Extruder(0.037)
  MoveL 390 to (511.12, 489.23, 0.3) mm, rotated rx 0 ry 90 rz 0 deg; joints [-10.822, -26.16, 109.68, -14.836, -82.872, 50.884]
  Call Extruder(0.038)
  MoveL 391 to (511.28, 489.52, 0.3) mm, rotated rx 0 ry 90 rz 0 deg; joints [-10.846, -26.156, 109.655, -14.861, -82.852, 50.892]
  Call Extruder(0.055)
  MoveL 392 to (511.37, 490, 0.3) mm, rotated rx 0 ry 90 rz 0 deg; joints [-10.888, -26.153, 109.634, -14.904, -82.836, 50.902]
  Call Extruder(2.270)
  MoveL 393 to (511.37, 510, 0.3) mm, rotated rx 0 ry 90 rz 0 deg; joints [-12.688, -26.073, 109.131, -16.733, -82.487, 51.222]
  Call Extruder(0.037)
  MoveL 394 to (511.32, 510.33, 0.3) mm, rotated rx 0 ry 90 rz 0 deg; joints [-12.718, -26.072, 109.127, -16.764, -82.485, 51.227]
  Call Extruder(0.037)
  MoveL 395 to (511.21, 510.64, 0.3) mm, rotated rx 0 ry 90 rz 0 deg; joints [-12.748, -26.073, 109.133, -16.794, -82.49, 51.229]
  Call Extruder(0.037)
  MoveL 396 to (511.02, 510.91, 0.3) mm, rotated rx 0 ry 90 rz 0 deg; joints [-12.777, -26.076, 109.148, -16.822, -82.504, 51.229]
  Call Extruder(0.037)
  MoveL 397 to (510.77, 511.12, 0.3) mm, rotated rx 0 ry 90 rz 0 deg; joints [-12.801, -26.079, 109.172, -16.846, -82.523, 51.226]
  Call Extruder(0.038)
  MoveL 398 to (510.48, 511.28, 0.3) mm, rotated rx 0 ry 90 rz 0 deg; joints [-12.821, -26.084, 109.203, -16.864, -82.549, 51.22]
  Call Extruder(0.055)
  MoveL 399 to (510, 511.37, 0.3) mm, rotated rx 0 ry 90 rz 0 deg; joints [-12.838, -26.093, 109.258, -16.88, -82.594, 51.209]
  Call Extruder(2.270)
  MoveL 400 to (490, 511.37, 0.3) mm, rotated rx 0 ry 90 rz 0 deg; joints [-13.259, -26.444, 111.632, -17.237, -84.541, 50.653]
  Call Extruder(0.037)
  MoveL 401 to (489.67, 511.33, 0.3) mm, rotated rx 0 ry 90 rz 0 deg; joints [-13.263, -26.449, 111.672, -17.24, -84.574, 50.643]
  Call Extruder(0.037)
  MoveL 402 to (489.36, 511.21, 0.3) mm, rotated rx 0 ry 90 rz 0 deg; joints [-13.259, -26.455, 111.711, -17.234, -84.606, 50.632]
  Call Extruder(0.037)
  MoveL 403 to (489.09, 511.02, 0.3) mm, rotated rx 0 ry 90 rz 0 deg; joints [-13.247, -26.46, 111.748, -17.222, -84.636, 50.622]
  Call Extruder(0.037)
  MoveL 404 to (488.87, 510.77, 0.3) mm, rotated rx 0 ry 90 rz 0 deg; joints [-13.229, -26.464, 111.78, -17.203, -84.663, 50.612]
  Call Extruder(0.038)
  MoveL 405 to (488.72, 510.48, 0.3) mm, rotated rx 0 ry 90 rz 0 deg; joints [-13.205, -26.467, 111.806, -17.179, -84.684, 50.603]
  Call Extruder(0.055)
  MoveL 406 to (488.63, 510, 0.3) mm, rotated rx 0 ry 90 rz 0 deg; joints [-13.163, -26.471, 111.83, -17.135, -84.702, 50.594]
  Call Extruder(2.270)
  MoveL 407 to (488.63, 490, 0.3) mm, rotated rx 0 ry 90 rz 0 deg; joints [-11.299, -26.536, 112.339, -15.253, -85.088, 50.332]
  Call Extruder(0.037)
  MoveL 408 to (488.67, 489.67, 0.3) mm, rotated rx 0 ry 90 rz 0 deg; joints [-11.267, -26.537, 112.342, -15.222, -85.089, 50.329]
  Call Extruder(0.037)
  MoveL 409 to (488.79, 489.36, 0.3) mm, rotated rx 0 ry 90 rz 0 deg; joints [-11.236, -26.536, 112.335, -15.19, -85.083, 50.328]
  Call Extruder(0.037)
  MoveL 410 to (488.98, 489.09, 0.3) mm, rotated rx 0 ry 90 rz 0 deg; joints [-11.207, -26.534, 112.319, -15.162, -85.069, 50.33]
  Set speed (60.0 mm/s)
  MoveL 411 to (489.7, 489.66, 0.3) mm, rotated rx 0 ry 90 rz 0 deg; joints [-11.247, -26.522, 112.222, -15.204, -84.988, 50.355]
  Set speed (15.0 mm/s)
  Call Extruder(0.022)
  MoveL 412 to (489.86, 489.57, 0.3) mm, rotated rx 0 ry 90 rz 0 deg; joints [-11.235, -26.519, 112.205, -15.192, -84.973, 50.358]
  Call Extruder(0.016)
  MoveL 413 to (490, 489.55, 0.3) mm, rotated rx 0 ry 90 rz 0 deg; joints [-11.23, -26.517, 112.189, -15.188, -84.96, 50.361]
  Call Extruder(2.270)
  MoveL 414 to (510, 489.55, 0.3) mm, rotated rx 0 ry 90 rz 0 deg; joints [-10.87, -26.18, 109.809, -14.882, -82.978, 50.861]
  Call Extruder(0.022)
  MoveL 415 to (510.19, 489.59, 0.3) mm, rotated rx 0 ry 90 rz 0 deg; joints [-10.871, -26.176, 109.785, -14.883, -82.959, 50.867]
  Call Extruder(0.021)
  MoveL 416 to (510.34, 489.7, 0.3) mm, rotated rx 0 ry 90 rz 0 deg; joints [-10.878, -26.173, 109.764, -14.891, -82.942, 50.872]
  Call Extruder(0.022)
  MoveL 417 to (510.43, 489.86, 0.3) mm, rotated rx 0 ry 90 rz 0 deg; joints [-10.891, -26.171, 109.749, -14.905, -82.93, 50.877]
  Call Extruder(0.016)
  MoveL 418 to (510.45, 490, 0.3) mm, rotated rx 0 ry 90 rz 0 deg; joints [-10.904, -26.17, 109.743, -14.917, -82.926, 50.879]
  Call Extruder(2.270)
  MoveL 419 to (510.45, 510, 0.3) mm, rotated rx 0 ry 90 rz 0 deg; joints [-12.707, -26.091, 109.24, -16.748, -82.575, 51.198]
  Call Extruder(0.022)
  MoveL 420 to (510.42, 510.19, 0.3) mm, rotated rx 0 ry 90 rz 0 deg; joints [-12.724, -26.09, 109.24, -16.766, -82.576, 51.2]
  Call Extruder(0.021)
  MoveL 421 to (510.3, 510.34, 0.3) mm, rotated rx 0 ry 90 rz 0 deg; joints [-12.74, -26.092, 109.249, -16.782, -82.584, 51.2]
  Call Extruder(0.022)
  MoveL 422 to (510.14, 510.43, 0.3) mm, rotated rx 0 ry 90 rz 0 deg; joints [-12.752, -26.095, 109.267, -16.793, -82.598, 51.197]
  Call Extruder(0.016)
  MoveL 423 to (510, 510.46, 0.3) mm, rotated rx 0 ry 90 rz 0 deg; joints [-12.757, -26.097, 109.283, -16.797, -82.611, 51.193]
  Call Extruder(2.270)
  MoveL 424 to (490, 510.46, 0.3) mm, rotated rx 0 ry 90 rz 0 deg; joints [-13.175, -26.448, 111.657, -17.152, -84.559, 50.639]
  Call Extruder(0.022)
  MoveL 425 to (489.81, 510.42, 0.3) mm, rotated rx 0 ry 90 rz 0 deg; joints [-13.176, -26.451, 111.68, -17.152, -84.578, 50.634]
  Call Extruder(0.021)
  MoveL 426 to (489.66, 510.3, 0.3) mm, rotated rx 0 ry 90 rz 0 deg; joints [-13.169, -26.453, 111.701, -17.144, -84.596, 50.628]
  Call Extruder(0.022)
  MoveL 427 to (489.57, 510.14, 0.3) mm, rotated rx 0 ry 90 rz 0 deg; joints [-13.156, -26.455, 111.717, -17.131, -84.608, 50.623]
  Call Extruder(0.016)
  MoveL 428 to (489.54, 510, 0.3) mm, rotated rx 0 ry 90 rz 0 deg; joints [-13.143, -26.456, 111.723, -17.118, -84.613, 50.62]
  Call Extruder(2.270)
  MoveL 429 to (489.54, 490, 0.3) mm, rotated rx 0 ry 90 rz 0 deg; joints [-11.282, -26.523, 112.232, -15.238, -84.997, 50.355]
  Call Extruder(0.022)
  MoveL 430 to (489.59, 489.81, 0.3) mm, rotated rx 0 ry 90 rz 0 deg; joints [-11.263, -26.523, 112.231, -15.22, -84.996, 50.354]
  Call Extruder(0.021)
  MoveL 431 to (489.7, 489.66, 0.3) mm, rotated rx 0 ry 90 rz 0 deg; joints [-11.247, -26.522, 112.222, -15.204, -84.988, 50.355]
  Set speed (30.0 mm/s)
  Call Extruder(-0.400)
  MoveL 432 to (489.7, 489.66, 0.3) mm, rotated rx 0 ry 90 rz 0 deg; joints [-11.247, -26.522, 112.222, -15.204, -84.988, 50.355]
  Set speed (60.0 mm/s)
  MoveL 433 to (490.61, 509.43, 0.3) mm, rotated rx 0 ry 90 rz 0 deg; joints [-13.067, -26.442, 111.614, -17.045, -84.521, 50.642]
  Set speed (1000.0 mm/s)
  MoveL 434 to (490.51, 509.5, 0.3) mm, rotated rx 0 ry 90 rz 0 deg; joints [-13.076, -26.443, 111.624, -17.053, -84.53, 50.64]
  Set speed (30.0 mm/s)
  Call Extruder(0.400)
  MoveL 435 to (490.51, 509.5, 0.3) mm, rotated rx 0 ry 90 rz 0 deg; joints [-13.076, -26.443, 111.624, -17.053, -84.53, 50.64]
  Set speed (15.0 mm/s)
  Call Extruder(2.155)
  MoveL 436 to (490.51, 490.51, 0.3) mm, rotated rx 0 ry 90 rz 0 deg; joints [-11.311, -26.507, 112.107, -15.27, -84.893, 50.386]
  MoveL 437 to (509.49, 490.5, 0.3) mm, rotated rx 0 ry 90 rz 0 deg; joints [-10.966, -26.186, 109.847, -14.977, -83.012, 50.863]
  MoveL 438 to (509.49, 509.5, 0.3) mm, rotated rx 0 ry 90 rz 0 deg; joints [-12.681, -26.111, 109.369, -16.718, -82.678, 51.163]
  MoveL 439 to (490.51, 509.5, 0.3) mm, rotated rx 0 ry 90 rz 0 deg; joints [-13.076, -26.443, 111.624, -17.053, -84.53, 50.64]
  Set speed (60.0 mm/s)
  MoveL 440 to (490.5, 509.1, 0.3) mm, rotated rx 0 ry 90 rz 0 deg; joints [-13.039, -26.445, 111.635, -17.016, -84.538, 50.634]
  Set speed (1000.0 mm/s)
  MoveL 441 to (490.6, 509.1, 0.3) mm, rotated rx 0 ry 90 rz 0 deg; joints [-13.037, -26.443, 111.623, -17.014, -84.528, 50.637]
  Set speed (1000.0 mm/s)
  MoveL 442 to (491.41, 508.6, 0.3) mm, rotated rx 0 ry 90 rz 0 deg; joints [-12.974, -26.432, 111.543, -16.952, -84.46, 50.652]
  Set speed (15.0 mm/s)
  Call Extruder(1.951)
  MoveL 443 to (491.4, 491.4, 0.3) mm, rotated rx 0 ry 90 rz 0 deg; joints [-11.378, -26.49, 111.98, -15.34, -84.787, 50.42]
  MoveL 444 to (508.6, 491.41, 0.3) mm, rotated rx 0 ry 90 rz 0 deg; joints [-11.064, -26.199, 109.934, -15.073, -83.086, 50.854]
  MoveL 445 to (508.59, 508.6, 0.3) mm, rotated rx 0 ry 90 rz 0 deg; joints [-12.618, -26.132, 109.502, -16.651, -82.783, 51.124]
  MoveL 446 to (491.41, 508.6, 0.3) mm, rotated rx 0 ry 90 rz 0 deg; joints [-12.974, -26.432, 111.543, -16.952, -84.46, 50.652]
  Set speed (60.0 mm/s)
  MoveL 447 to (492.73, 508.17, 0.3) mm, rotated rx 0 ry 90 rz 0 deg; joints [-12.907, -26.412, 111.398, -16.889, -84.339, 50.683]
  Set speed (15.0 mm/s)
  Call Extruder(0.146)
  MoveL 448 to (491.82, 507.27, 0.3) mm, rotated rx 0 ry 90 rz 0 deg; joints [-12.842, -26.43, 111.529, -16.821, -84.446, 50.645]
  Set speed (60.0 mm/s)
  MoveL 449 to (491.82, 505.98, 0.3) mm, rotated rx 0 ry 90 rz 0 deg; joints [-12.724, -26.435, 111.564, -16.701, -84.471, 50.626]
  Set speed (15.0 mm/s)
  Call Extruder(0.352)
  MoveL 450 to (494.02, 508.17, 0.3) mm, rotated rx 0 ry 90 rz 0 deg; joints [-12.88, -26.391, 111.246, -16.865, -84.213, 50.719]
  Set speed (60.0 mm/s)
  MoveL 451 to (495.3, 508.17, 0.3) mm, rotated rx 0 ry 90 rz 0 deg; joints [-12.853, -26.37, 111.095, -16.842, -84.087, 50.755]
  Set speed (15.0 mm/s)
  Call Extruder(0.559)
  MoveL 452 to (491.82, 504.69, 0.3) mm, rotated rx 0 ry 90 rz 0 deg; joints [-12.605, -26.439, 111.598, -16.58, -84.496, 50.608]
  Set speed (60.0 mm/s)
  MoveL 453 to (491.82, 503.41, 0.3) mm, rotated rx 0 ry 90 rz 0 deg; joints [-12.486, -26.444, 111.631, -16.46, -84.522, 50.59]
  Set speed (15.0 mm/s)
  Call Extruder(0.765)
  MoveL 454 to (496.59, 508.17, 0.3) mm, rotated rx 0 ry 90 rz 0 deg; joints [-12.826, -26.349, 110.942, -16.819, -83.962, 50.79]
  Set speed (60.0 mm/s)
  MoveL 455 to (497.88, 508.17, 0.3) mm, rotated rx 0 ry 90 rz 0 deg; joints [-12.799, -26.327, 110.79, -16.796, -83.836, 50.826]
  Set speed (15.0 mm/s)
  Call Extruder(0.972)
  MoveL 456 to (491.82, 502.12, 0.3) mm, rotated rx 0 ry 90 rz 0 deg; joints [-12.366, -26.449, 111.665, -16.34, -84.546, 50.573]
  Set speed (60.0 mm/s)
  MoveL 457 to (491.82, 500.83, 0.3) mm, rotated rx 0 ry 90 rz 0 deg; joints [-12.247, -26.453, 111.698, -16.219, -84.571, 50.555]
  Set speed (15.0 mm/s)
  Call Extruder(1.178)
  MoveL 458 to (499.16, 508.17, 0.3) mm, rotated rx 0 ry 90 rz 0 deg; joints [-12.772, -26.305, 110.638, -16.773, -83.71, 50.861]
  Set speed (60.0 mm/s)
  MoveL 459 to (500.45, 508.17, 0.3) mm, rotated rx 0 ry 90 rz 0 deg; joints [-12.746, -26.282, 110.485, -16.751, -83.585, 50.896]
  Set speed (15.0 mm/s)
  Call Extruder(1.385)
  MoveL 460 to (491.82, 499.55, 0.3) mm, rotated rx 0 ry 90 rz 0 deg; joints [-12.128, -26.457, 111.731, -16.098, -84.596, 50.537]
  Set speed (60.0 mm/s)
  MoveL 461 to (491.82, 498.26, 0.3) mm, rotated rx 0 ry 90 rz 0 deg; joints [-12.008, -26.462, 111.763, -15.978, -84.62, 50.52]
  Set speed (15.0 mm/s)
  Call Extruder(1.591)
  MoveL 462 to (501.74, 508.17, 0.3) mm, rotated rx 0 ry 90 rz 0 deg; joints [-12.719, -26.259, 110.332, -16.729, -83.459, 50.932]
  Set speed (60.0 mm/s)
  MoveL 463 to (503.03, 508.17, 0.3) mm, rotated rx 0 ry 90 rz 0 deg; joints [-12.693, -26.237, 110.178, -16.706, -83.333, 50.967]
  Set speed (15.0 mm/s)
  Call Extruder(1.798)
  MoveL 464 to (491.82, 496.97, 0.3) mm, rotated rx 0 ry 90 rz 0 deg; joints [-11.889, -26.466, 111.795, -15.857, -84.644, 50.503]
  Set speed (60.0 mm/s)
  MoveL 465 to (491.82, 495.69, 0.3) mm, rotated rx 0 ry 90 rz 0 deg; joints [-11.769, -26.47, 111.827, -15.736, -84.668, 50.486]
  Set speed (15.0 mm/s)
  Call Extruder(2.005)
  MoveL 466 to (504.31, 508.17, 0.3) mm, rotated rx 0 ry 90 rz 0 deg; joints [-12.667, -26.213, 110.025, -16.684, -83.208, 51.002]
  Set speed (60.0 mm/s)
  MoveL 467 to (505.6, 508.17, 0.3) mm, rotated rx 0 ry 90 rz 0 deg; joints [-12.641, -26.19, 109.871, -16.663, -83.082, 51.037]
  Set speed (15.0 mm/s)
  Call Extruder(2.211)
  MoveL 468 to (491.82, 494.4, 0.3) mm, rotated rx 0 ry 90 rz 0 deg; joints [-11.649, -26.474, 111.858, -15.615, -84.691, 50.469]
  Set speed (60.0 mm/s)
  MoveL 469 to (491.82, 493.11, 0.3) mm, rotated rx 0 ry 90 rz 0 deg; joints [-11.529, -26.478, 111.889, -15.494, -84.715, 50.453]
  Set speed (15.0 mm/s)
  Call Extruder(2.418)
  MoveL 470 to (506.89, 508.17, 0.3) mm, rotated rx 0 ry 90 rz 0 deg; joints [-12.615, -26.166, 109.717, -16.641, -82.957, 51.071]
  Set speed (60.0 mm/s)
  MoveL 471 to (508.17, 508.17, 0.3) mm, rotated rx 0 ry 90 rz 0 deg; joints [-12.589, -26.142, 109.563, -16.62, -82.832, 51.106]
  Set speed (15.0 mm/s)
  Call Extruder(2.624)
  MoveL 472 to (491.82, 491.82, 0.3) mm, rotated rx 0 ry 90 rz 0 deg; joints [-11.409, -26.482, 111.92, -15.373, -84.738, 50.436]
  Set speed (60.0 mm/s)
  MoveL 473 to (493.11, 491.82, 0.3) mm, rotated rx 0 ry 90 rz 0 deg; joints [-11.385, -26.462, 111.768, -15.352, -84.611, 50.47]
  Set speed (15.0 mm/s)
  Call Extruder(2.418)
  MoveL 474 to (508.17, 506.89, 0.3) mm, rotated rx 0 ry 90 rz 0 deg; joints [-12.473, -26.147, 109.598, -16.502, -82.856, 51.085]
  Set speed (60.0 mm/s)
  MoveL 475 to (508.17, 505.6, 0.3) mm, rotated rx 0 ry 90 rz 0 deg; joints [-12.357, -26.152, 109.632, -16.384, -82.879, 51.064]
  Set speed (15.0 mm/s)
  Call Extruder(2.211)
  MoveL 476 to (494.4, 491.82, 0.3) mm, rotated rx 0 ry 90 rz 0 deg; joints [-11.361, -26.442, 111.616, -15.331, -84.483, 50.503]
  Set speed (60.0 mm/s)
  MoveL 477 to (495.68, 491.82, 0.3) mm, rotated rx 0 ry 90 rz 0 deg; joints [-11.337, -26.421, 111.464, -15.31, -84.356, 50.536]
  Set speed (15.0 mm/s)
  Call Extruder(2.005)
  MoveL 478 to (508.17, 504.31, 0.3) mm, rotated rx 0 ry 90 rz 0 deg; joints [-12.241, -26.158, 109.665, -16.266, -82.903, 51.043]
  Set speed (60.0 mm/s)
  MoveL 479 to (508.17, 503.03, 0.3) mm, rotated rx 0 ry 90 rz 0 deg; joints [-12.125, -26.163, 109.698, -16.148, -82.926, 51.023]
  Set speed (15.0 mm/s)
  Call Extruder(1.798)
  MoveL 480 to (496.97, 491.82, 0.3) mm, rotated rx 0 ry 90 rz 0 deg; joints [-11.313, -26.4, 111.311, -15.29, -84.228, 50.568]
  Set speed (60.0 mm/s)
  MoveL 481 to (498.26, 491.82, 0.3) mm, rotated rx 0 ry 90 rz 0 deg; joints [-11.29, -26.379, 111.159, -15.27, -84.101, 50.601]
  Set speed (15.0 mm/s)
  Call Extruder(1.591)
  MoveL 482 to (508.17, 501.74, 0.3) mm, rotated rx 0 ry 90 rz 0 deg; joints [-12.009, -26.168, 109.731, -16.03, -82.949, 51.002]
  Set speed (60.0 mm/s)
  MoveL 483 to (508.17, 500.45, 0.3) mm, rotated rx 0 ry 90 rz 0 deg; joints [-11.892, -26.173, 109.764, -15.912, -82.972, 50.982]
  Set speed (15.0 mm/s)
  Call Extruder(1.385)
  MoveL 484 to (499.55, 491.82, 0.3) mm, rotated rx 0 ry 90 rz 0 deg; joints [-11.266, -26.358, 111.006, -15.249, -83.973, 50.634]
  Set speed (60.0 mm/s)
  MoveL 485 to (500.83, 491.82, 0.3) mm, rotated rx 0 ry 90 rz 0 deg; joints [-11.242, -26.336, 110.853, -15.229, -83.846, 50.666]
  Set speed (15.0 mm/s)
  Call Extruder(1.178)
  MoveL 486 to (508.17, 499.16, 0.3) mm, rotated rx 0 ry 90 rz 0 deg; joints [-11.776, -26.178, 109.797, -15.794, -82.995, 50.962]
  Set speed (60.0 mm/s)
  MoveL 487 to (508.17, 497.88, 0.3) mm, rotated rx 0 ry 90 rz 0 deg; joints [-11.659, -26.183, 109.829, -15.676, -83.018, 50.942]
  Set speed (15.0 mm/s)
  Call Extruder(0.972)
  MoveL 488 to (502.12, 491.82, 0.3) mm, rotated rx 0 ry 90 rz 0 deg; joints [-11.219, -26.314, 110.699, -15.209, -83.719, 50.699]
  Set speed (60.0 mm/s)
  MoveL 489 to (503.41, 491.82, 0.3) mm, rotated rx 0 ry 90 rz 0 deg; joints [-11.195, -26.291, 110.546, -15.19, -83.592, 50.731]
  Set speed (15.0 mm/s)
  Call Extruder(0.765)
  MoveL 490 to (508.17, 496.59, 0.3) mm, rotated rx 0 ry 90 rz 0 deg; joints [-11.543, -26.188, 109.86, -15.557, -83.04, 50.922]
  Set speed (60.0 mm/s)
  MoveL 491 to (508.17, 495.3, 0.3) mm, rotated rx 0 ry 90 rz 0 deg; joints [-11.426, -26.193, 109.892, -15.439, -83.062, 50.902]
  Set speed (15.0 mm/s)
  Call Extruder(0.559)
  MoveL 492 to (504.69, 491.82, 0.3) mm, rotated rx 0 ry 90 rz 0 deg; joints [-11.172, -26.268, 110.392, -15.17, -83.465, 50.763]
  Set speed (60.0 mm/s)
  MoveL 493 to (505.98, 491.82, 0.3) mm, rotated rx 0 ry 90 rz 0 deg; joints [-11.149, -26.245, 110.238, -15.151, -83.338, 50.796]
  Set speed (15.0 mm/s)
  Call Extruder(0.352)
  MoveL 494 to (508.17, 494.02, 0.3) mm, rotated rx 0 ry 90 rz 0 deg; joints [-11.309, -26.198, 109.923, -15.32, -83.084, 50.883]
  Set speed (60.0 mm/s)
  MoveL 495 to (508.17, 492.73, 0.3) mm, rotated rx 0 ry 90 rz 0 deg; joints [-11.192, -26.202, 109.953, -15.202, -83.106, 50.864]
  Set speed (15.0 mm/s)
  Call Extruder(0.146)
  MoveL 496 to (507.27, 491.82, 0.3) mm, rotated rx 0 ry 90 rz 0 deg; joints [-11.126, -26.222, 110.084, -15.132, -83.21, 50.828]
  Set speed (60.0 mm/s)
  MoveL 497 to (490.58, 509.43, 0.3) mm, rotated rx 0 ry 90 rz 0 deg; joints [-13.068, -26.442, 111.618, -17.045, -84.524, 50.641]
  Set speed (1000.0 mm/s)
  MoveL 498 to (490.4, 509.6, 0.3) mm, rotated rx 0 ry 90 rz 0 deg; joints [-13.088, -26.444, 111.634, -17.065, -84.538, 50.638]
  Call M_RunCode(106)
  Call SetRPM(255.0)
  Set speed (90.0 mm/s)
  MoveL 499 to (490.4, 509.6, 0.4) mm, rotated rx 0 ry 90 rz 0 deg; joints [-13.088, -26.455, 111.639, -17.065, -84.533, 50.64]
  Set speed (15.0 mm/s)
  Call Extruder(0.559)
  MoveL 500 to (490.4, 490.4, 0.4) mm, rotated rx 0 ry 90 rz 0 deg; joints [-11.303, -26.519, 112.127, -15.262, -84.9, 50.383]
  MoveL 501 to (509.6, 490.4, 0.4) mm, rotated rx 0 ry 90 rz 0 deg; joints [-10.955, -26.195, 109.842, -14.966, -82.999, 50.866]
  MoveL 502 to (509.6, 509.6, 0.4) mm, rotated rx 0 ry 90 rz 0 deg; joints [-12.688, -26.119, 109.359, -16.726, -82.661, 51.17]
  MoveL 503 to (490.4, 509.6, 0.4) mm, rotated rx 0 ry 90 rz 0 deg; joints [-13.088, -26.455, 111.639, -17.065, -84.533, 50.64]
  Set speed (90.0 mm/s)
  MoveL 504 to (490.4, 509.2, 0.4) mm, rotated rx 0 ry 90 rz 0 deg; joints [-13.051, -26.456, 111.65, -17.028, -84.541, 50.634]
  Set speed (1000.0 mm/s)
  MoveL 505 to (491.09, 508.91, 0.4) mm, rotated rx 0 ry 90 rz 0 deg; joints [-13.01, -26.447, 111.577, -16.988, -84.479, 50.649]
  Set speed (15.0 mm/s)
  Call Extruder(0.519)
  MoveL 506 to (491.09, 491.09, 0.4) mm, rotated rx 0 ry 90 rz 0 deg; joints [-11.355, -26.507, 112.03, -15.316, -84.819, 50.41]
  MoveL 507 to (508.91, 491.09, 0.4) mm, rotated rx 0 ry 90 rz 0 deg; joints [-11.03, -26.205, 109.909, -15.04, -83.056, 50.859]
  MoveL 508 to (508.91, 508.91, 0.4) mm, rotated rx 0 ry 90 rz 0 deg; joints [-12.64, -26.135, 109.461, -16.675, -82.741, 51.139]
  MoveL 509 to (491.09, 508.91, 0.4) mm, rotated rx 0 ry 90 rz 0 deg; joints [-13.01, -26.447, 111.577, -16.988, -84.479, 50.649]
  Set speed (90.0 mm/s)
  MoveL 510 to (491.4, 491.62, 0.4) mm, rotated rx 0 ry 90 rz 0 deg; joints [-11.398, -26.5, 111.98, -15.36, -84.779, 50.424]
  Set speed (15.0 mm/s)
  Call Extruder(0.009)
  MoveL 511 to (491.62, 491.4, 0.4) mm, rotated rx 0 ry 90 rz 0 deg; joints [-11.374, -26.498, 111.96, -15.337, -84.761, 50.427]
  Set speed (90.0 mm/s)
  MoveL 512 to (492.61, 491.4, 0.4) mm, rotated rx 0 ry 90 rz 0 deg; joints [-11.356, -26.482, 111.844, -15.321, -84.663, 50.453]
  Set speed (15.0 mm/s)
  Call Extruder(0.049)
  MoveL 513 to (491.4, 492.61, 0.4) mm, rotated rx 0 ry 90 rz 0 deg; joints [-11.49, -26.497, 111.957, -15.454, -84.761, 50.437]
  Set speed (90.0 mm/s)
  MoveL 514 to (491.4, 493.6, 0.4) mm, rotated rx 0 ry 90 rz 0 deg; joints [-11.583, -26.494, 111.933, -15.547, -84.743, 50.449]
  Set speed (15.0 mm/s)
  Call Extruder(0.090)
  MoveL 515 to (493.6, 491.4, 0.4) mm, rotated rx 0 ry 90 rz 0 deg; joints [-11.337, -26.467, 111.727, -15.305, -84.565, 50.478]
  Set speed (90.0 mm/s)
  MoveL 516 to (494.58, 491.4, 0.4) mm, rotated rx 0 ry 90 rz 0 deg; joints [-11.319, -26.451, 111.61, -15.289, -84.467, 50.503]
  Set speed (15.0 mm/s)
  Call Extruder(0.131)
  MoveL 517 to (491.4, 494.59, 0.4) mm, rotated rx 0 ry 90 rz 0 deg; joints [-11.675, -26.491, 111.909, -15.64, -84.725, 50.462]
  Set speed (90.0 mm/s)
  MoveL 518 to (491.4, 495.58, 0.4) mm, rotated rx 0 ry 90 rz 0 deg; joints [-11.767, -26.488, 111.885, -15.733, -84.706, 50.475]
  Set speed (15.0 mm/s)
  Call Extruder(0.172)
  MoveL 519 to (495.57, 491.4, 0.4) mm, rotated rx 0 ry 90 rz 0 deg; joints [-11.3, -26.435, 111.492, -15.273, -84.369, 50.529]
  Set speed (90.0 mm/s)
  MoveL 520 to (496.57, 491.4, 0.4) mm, rotated rx 0 ry 90 rz 0 deg; joints [-11.282, -26.419, 111.375, -15.257, -84.271, 50.554]
  Set speed (15.0 mm/s)
  Call Extruder(0.212)
  MoveL 521 to (491.4, 496.56, 0.4) mm, rotated rx 0 ry 90 rz 0 deg; joints [-11.859, -26.484, 111.86, -15.826, -84.688, 50.488]
  Set speed (90.0 mm/s)
  MoveL 522 to (491.4, 497.55, 0.4) mm, rotated rx 0 ry 90 rz 0 deg; joints [-11.951, -26.481, 111.836, -15.919, -84.67, 50.501]
  Set speed (15.0 mm/s)
  Call Extruder(0.253)
  MoveL 523 to (497.55, 491.4, 0.4) mm, rotated rx 0 ry 90 rz 0 deg; joints [-11.264, -26.403, 111.258, -15.242, -84.173, 50.579]
  Set speed (90.0 mm/s)
  MoveL 524 to (498.54, 491.4, 0.4) mm, rotated rx 0 ry 90 rz 0 deg; joints [-11.245, -26.386, 111.14, -15.226, -84.075, 50.604]
  Set speed (15.0 mm/s)
  Call Extruder(0.294)
  MoveL 525 to (491.4, 498.54, 0.4) mm, rotated rx 0 ry 90 rz 0 deg; joints [-12.043, -26.478, 111.811, -16.012, -84.651, 50.514]
  Set speed (90.0 mm/s)
  MoveL 526 to (491.4, 499.53, 0.4) mm, rotated rx 0 ry 90 rz 0 deg; joints [-12.135, -26.475, 111.786, -16.105, -84.632, 50.527]
  Set speed (15.0 mm/s)
  Call Extruder(0.335)
  MoveL 527 to (499.53, 491.4, 0.4) mm, rotated rx 0 ry 90 rz 0 deg; joints [-11.227, -26.37, 111.023, -15.211, -83.977, 50.629]
  Set speed (90.0 mm/s)
  MoveL 528 to (500.52, 491.4, 0.4) mm, rotated rx 0 ry 90 rz 0 deg; joints [-11.209, -26.353, 110.905, -15.195, -83.879, 50.654]
  Set speed (15.0 mm/s)
  Call Extruder(0.375)
  MoveL 529 to (491.4, 500.52, 0.4) mm, rotated rx 0 ry 90 rz 0 deg; joints [-12.227, -26.471, 111.761, -16.198, -84.613, 50.541]
  Set speed (90.0 mm/s)
  MoveL 530 to (491.4, 501.51, 0.4) mm, rotated rx 0 ry 90 rz 0 deg; joints [-12.319, -26.468, 111.735, -16.29, -84.594, 50.554]
  Set speed (15.0 mm/s)
  Call Extruder(0.416)
  MoveL 531 to (501.51, 491.4, 0.4) mm, rotated rx 0 ry 90 rz 0 deg; joints [-11.191, -26.336, 110.787, -15.18, -83.781, 50.679]
  Set speed (90.0 mm/s)
  MoveL 532 to (502.5, 491.4, 0.4) mm, rotated rx 0 ry 90 rz 0 deg; joints [-11.173, -26.319, 110.669, -15.165, -83.683, 50.704]
  Set speed (15.0 mm/s)
  Call Extruder(0.457)
  MoveL 533 to (491.4, 502.5, 0.4) mm, rotated rx 0 ry 90 rz 0 deg; joints [-12.411, -26.464, 111.71, -16.383, -84.575, 50.568]
  Set speed (90.0 mm/s)
  MoveL 534 to (491.4, 503.49, 0.4) mm, rotated rx 0 ry 90 rz 0 deg; joints [-12.502, -26.461, 111.684, -16.476, -84.556, 50.582]
  Set speed (15.0 mm/s)
  Call Extruder(0.498)
  MoveL 535 to (503.49, 491.4, 0.4) mm, rotated rx 0 ry 90 rz 0 deg; joints [-11.155, -26.302, 110.551, -15.15, -83.585, 50.729]
  Set speed (90.0 mm/s)
  MoveL 536 to (504.48, 491.4, 0.4) mm, rotated rx 0 ry 90 rz 0 deg; joints [-11.137, -26.284, 110.432, -15.135, -83.487, 50.754]
  Set speed (15.0 mm/s)
  Call Extruder(0.538)
  MoveL 537 to (491.4, 504.48, 0.4) mm, rotated rx 0 ry 90 rz 0 deg; joints [-12.594, -26.458, 111.658, -16.568, -84.537, 50.595]
  Set speed (90.0 mm/s)
  MoveL 538 to (491.4, 505.47, 0.4) mm, rotated rx 0 ry 90 rz 0 deg; joints [-12.686, -26.454, 111.632, -16.661, -84.517, 50.609]
  Set speed (15.0 mm/s)
  Call Extruder(0.579)
  MoveL 539 to (505.47, 491.4, 0.4) mm, rotated rx 0 ry 90 rz 0 deg; joints [-11.12, -26.267, 110.314, -15.12, -83.39, 50.778]
  Set speed (90.0 mm/s)
  MoveL 540 to (506.46, 491.4, 0.4) mm, rotated rx 0 ry 90 rz 0 deg; joints [-11.102, -26.249, 110.195, -15.105, -83.292, 50.803]
  Set speed (15.0 mm/s)
  Call Extruder(0.620)
  MoveL 541 to (491.4, 506.46, 0.4) mm, rotated rx 0 ry 90 rz 0 deg; joints [-12.777, -26.45, 111.606, -16.754, -84.498, 50.623]
  Set speed (90.0 mm/s)
  MoveL 542 to (491.4, 507.45, 0.4) mm, rotated rx 0 ry 90 rz 0 deg; joints [-12.868, -26.447, 111.579, -16.846, -84.478, 50.637]
  Set speed (15.0 mm/s)
  Call Extruder(0.661)
  MoveL 543 to (507.45, 491.4, 0.4) mm, rotated rx 0 ry 90 rz 0 deg; joints [-11.084, -26.231, 110.077, -15.09, -83.194, 50.828]
  Set speed (90.0 mm/s)
  MoveL 544 to (508.44, 491.4, 0.4) mm, rotated rx 0 ry 90 rz 0 deg; joints [-11.067, -26.213, 109.958, -15.076, -83.096, 50.852]
  Set speed (15.0 mm/s)
  Call Extruder(0.701)
  MoveL 545 to (491.4, 508.44, 0.4) mm, rotated rx 0 ry 90 rz 0 deg; joints [-12.96, -26.443, 111.552, -16.938, -84.458, 50.651]
  Set speed (90.0 mm/s)
  MoveL 546 to (492.24, 508.59, 0.4) mm, rotated rx 0 ry 90 rz 0 deg; joints [-12.956, -26.429, 111.45, -16.937, -84.373, 50.677]
  Set speed (15.0 mm/s)
  Call Extruder(0.673)
  MoveL 547 to (508.59, 492.24, 0.4) mm, rotated rx 0 ry 90 rz 0 deg; joints [-11.14, -26.207, 109.92, -15.151, -83.068, 50.868]
  Set speed (90.0 mm/s)
  MoveL 548 to (508.59, 493.23, 0.4) mm, rotated rx 0 ry 90 rz 0 deg; joints [-11.23, -26.203, 109.896, -15.242, -83.051, 50.883]
  Set speed (15.0 mm/s)
  Call Extruder(0.632)
  MoveL 549 to (493.23, 508.59, 0.4) mm, rotated rx 0 ry 90 rz 0 deg; joints [-12.935, -26.413, 111.333, -16.919, -84.276, 50.705]
  Set speed (90.0 mm/s)
  MoveL 550 to (494.22, 508.59, 0.4) mm, rotated rx 0 ry 90 rz 0 deg; joints [-12.914, -26.397, 111.216, -16.901, -84.18, 50.732]
  Set speed (15.0 mm/s)
  Call Extruder(0.591)
  MoveL 551 to (508.59, 494.22, 0.4) mm, rotated rx 0 ry 90 rz 0 deg; joints [-11.32, -26.2, 109.873, -15.333, -83.034, 50.898]
  Set speed (90.0 mm/s)
  MoveL 552 to (508.59, 495.21, 0.4) mm, rotated rx 0 ry 90 rz 0 deg; joints [-11.41, -26.196, 109.849, -15.424, -83.017, 50.913]
  Set speed (15.0 mm/s)
  Call Extruder(0.551)
  MoveL 553 to (495.21, 508.59, 0.4) mm, rotated rx 0 ry 90 rz 0 deg; joints [-12.893, -26.381, 111.099, -16.883, -84.083, 50.76]
  Set speed (90.0 mm/s)
  MoveL 554 to (496.2, 508.59, 0.4) mm, rotated rx 0 ry 90 rz 0 deg; joints [-12.872, -26.364, 110.982, -16.865, -83.986, 50.787]
  Set speed (15.0 mm/s)
  Call Extruder(0.510)
  MoveL 555 to (508.59, 496.2, 0.4) mm, rotated rx 0 ry 90 rz 0 deg; joints [-11.5, -26.192, 109.825, -15.515, -83, 50.928]
  Set speed (90.0 mm/s)
  MoveL 556 to (508.59, 497.19, 0.4) mm, rotated rx 0 ry 90 rz 0 deg; joints [-11.589, -26.188, 109.8, -15.606, -82.983, 50.943]
  Set speed (15.0 mm/s)
  Call Extruder(0.469)
  MoveL 557 to (497.19, 508.59, 0.4) mm, rotated rx 0 ry 90 rz 0 deg; joints [-12.852, -26.347, 110.865, -16.847, -83.89, 50.815]
  Set speed (90.0 mm/s)
  MoveL 558 to (498.18, 508.59, 0.4) mm, rotated rx 0 ry 90 rz 0 deg; joints [-12.831, -26.33, 110.748, -16.83, -83.793, 50.842]
  Set speed (15.0 mm/s)
  Call Extruder(0.428)
  MoveL 559 to (508.59, 498.18, 0.4) mm, rotated rx 0 ry 90 rz 0 deg; joints [-11.679, -26.185, 109.776, -15.697, -82.966, 50.959]
  Set speed (90.0 mm/s)
  MoveL 560 to (508.59, 499.17, 0.4) mm, rotated rx 0 ry 90 rz 0 deg; joints [-11.769, -26.181, 109.751, -15.788, -82.949, 50.974]
  Set speed (15.0 mm/s)
  Call Extruder(0.388)
  MoveL 561 to (499.17, 508.59, 0.4) mm, rotated rx 0 ry 90 rz 0 deg; joints [-12.811, -26.313, 110.631, -16.812, -83.696, 50.869]
  Set speed (90.0 mm/s)
  MoveL 562 to (500.16, 508.59, 0.4) mm, rotated rx 0 ry 90 rz 0 deg; joints [-12.79, -26.296, 110.513, -16.795, -83.6, 50.897]
  Set speed (15.0 mm/s)
  Call Extruder(0.347)
  MoveL 563 to (508.59, 500.16, 0.4) mm, rotated rx 0 ry 90 rz 0 deg; joints [-11.858, -26.177, 109.726, -15.879, -82.931, 50.99]
  Set speed (90.0 mm/s)
  MoveL 564 to (508.59, 501.15, 0.4) mm, rotated rx 0 ry 90 rz 0 deg; joints [-11.948, -26.173, 109.701, -15.97, -82.914, 51.005]
  Set speed (15.0 mm/s)
  Call Extruder(0.306)
  MoveL 565 to (501.15, 508.59, 0.4) mm, rotated rx 0 ry 90 rz 0 deg; joints [-12.77, -26.279, 110.395, -16.778, -83.503, 50.924]
  Set speed (90.0 mm/s)
  MoveL 566 to (502.14, 508.59, 0.4) mm, rotated rx 0 ry 90 rz 0 deg; joints [-12.749, -26.261, 110.278, -16.76, -83.407, 50.951]
  Set speed (15.0 mm/s)
  Call Extruder(0.265)
  MoveL 567 to (508.59, 502.14, 0.4) mm, rotated rx 0 ry 90 rz 0 deg; joints [-12.037, -26.169, 109.676, -16.061, -82.896, 51.021]
  Set speed (90.0 mm/s)
  MoveL 568 to (508.59, 503.13, 0.4) mm, rotated rx 0 ry 90 rz 0 deg; joints [-12.126, -26.165, 109.651, -16.152, -82.878, 51.037]
  Set speed (15.0 mm/s)
  Call Extruder(0.225)
  MoveL 569 to (503.13, 508.59, 0.4) mm, rotated rx 0 ry 90 rz 0 deg; joints [-12.729, -26.243, 110.16, -16.743, -83.31, 50.978]
  Set speed (90.0 mm/s)
  MoveL 570 to (504.12, 508.59, 0.4) mm, rotated rx 0 ry 90 rz 0 deg; joints [-12.709, -26.225, 110.042, -16.726, -83.214, 51.005]
  Set speed (15.0 mm/s)
  Call Extruder(0.184)
  MoveL 571 to (508.59, 504.12, 0.4) mm, rotated rx 0 ry 90 rz 0 deg; joints [-12.216, -26.161, 109.625, -16.242, -82.86, 51.053]
  Set speed (90.0 mm/s)
  MoveL 572 to (508.59, 505.11, 0.4) mm, rotated rx 0 ry 90 rz 0 deg; joints [-12.305, -26.157, 109.599, -16.333, -82.842, 51.069]
  Set speed (15.0 mm/s)
  Call Extruder(0.143)
  MoveL 573 to (505.11, 508.59, 0.4) mm, rotated rx 0 ry 90 rz 0 deg; joints [-12.689, -26.207, 109.924, -16.71, -83.117, 51.032]
  Set speed (90.0 mm/s)
  MoveL 574 to (506.1, 508.59, 0.4) mm, rotated rx 0 ry 90 rz 0 deg; joints [-12.668, -26.189, 109.805, -16.693, -83.021, 51.058]
  Set speed (15.0 mm/s)
  Call Extruder(0.103)
  MoveL 575 to (508.59, 506.1, 0.4) mm, rotated rx 0 ry 90 rz 0 deg; joints [-12.394, -26.153, 109.573, -16.423, -82.824, 51.085]
  Set speed (90.0 mm/s)
  MoveL 576 to (508.59, 507.09, 0.4) mm, rotated rx 0 ry 90 rz 0 deg; joints [-12.483, -26.149, 109.547, -16.514, -82.806, 51.101]
  Set speed (15.0 mm/s)
  Call Extruder(0.062)
  MoveL 577 to (507.09, 508.59, 0.4) mm, rotated rx 0 ry 90 rz 0 deg; joints [-12.648, -26.171, 109.687, -16.676, -82.924, 51.085]
  Set speed (90.0 mm/s)
  MoveL 578 to (508.08, 508.59, 0.4) mm, rotated rx 0 ry 90 rz 0 deg; joints [-12.628, -26.152, 109.568, -16.66, -82.828, 51.112]
  Set speed (15.0 mm/s)
  Call Extruder(0.021)
  MoveL 579 to (508.59, 508.08, 0.4) mm, rotated rx 0 ry 90 rz 0 deg; joints [-12.572, -26.145, 109.521, -16.604, -82.787, 51.117]
  Set speed (90.0 mm/s)
  MoveL 580 to (490.47, 509.53, 0.4) mm, rotated rx 0 ry 90 rz 0 deg; joints [-13.08, -26.454, 111.633, -17.057, -84.527, 50.641]
  Set speed (1000.0 mm/s)
  MoveL 581 to (490.4, 509.6, 0.4) mm, rotated rx 0 ry 90 rz 0 deg; joints [-13.088, -26.455, 111.639, -17.065, -84.533, 50.64]
  Set speed (120.0 mm/s)
  MoveL 582 to (490.4, 509.6, 0.5) mm, rotated rx 0 ry 90 rz 0 deg; joints [-13.088, -26.466, 111.644, -17.065, -84.528, 50.641]
  Set speed (15.0 mm/s)
  Call Extruder(0.559)
  MoveL 583 to (490.4, 490.4, 0.5) mm, rotated rx 0 ry 90 rz 0 deg; joints [-11.303, -26.53, 112.133, -15.262, -84.895, 50.385]
  MoveL 584 to (509.6, 490.4, 0.5) mm, rotated rx 0 ry 90 rz 0 deg; joints [-10.955, -26.205, 109.848, -14.966, -82.994, 50.867]
  MoveL 585 to (509.6, 509.6, 0.5) mm, rotated rx 0 ry 90 rz 0 deg; joints [-12.688, -26.13, 109.365, -16.726, -82.656, 51.171]
  MoveL 586 to (490.4, 509.6, 0.5) mm, rotated rx 0 ry 90 rz 0 deg; joints [-13.088, -26.466, 111.644, -17.065, -84.528, 50.641]
  Set speed (120.0 mm/s)
  MoveL 587 to (490.4, 509.2, 0.5) mm, rotated rx 0 ry 90 rz 0 deg; joints [-13.051, -26.467, 111.655, -17.028, -84.536, 50.636]
  Set speed (1000.0 mm/s)
  MoveL 588 to (491.09, 508.91, 0.5) mm, rotated rx 0 ry 90 rz 0 deg; joints [-13.01, -26.457, 111.582, -16.988, -84.474, 50.651]
  Set speed (15.0 mm/s)
  Call Extruder(0.519)
  MoveL 589 to (491.09, 491.09, 0.5) mm, rotated rx 0 ry 90 rz 0 deg; joints [-11.355, -26.517, 112.035, -15.316, -84.814, 50.411]
  MoveL 590 to (508.91, 491.09, 0.5) mm, rotated rx 0 ry 90 rz 0 deg; joints [-11.03, -26.216, 109.914, -15.04, -83.051, 50.86]
  MoveL 591 to (508.91, 508.91, 0.5) mm, rotated rx 0 ry 90 rz 0 deg; joints [-12.64, -26.146, 109.466, -16.675, -82.736, 51.141]
  MoveL 592 to (491.09, 508.91, 0.5) mm, rotated rx 0 ry 90 rz 0 deg; joints [-13.01, -26.457, 111.582, -16.988, -84.474, 50.651]
  Set speed (120.0 mm/s)
  MoveL 593 to (491.77, 508.59, 0.5) mm, rotated rx 0 ry 90 rz 0 deg; joints [-12.966, -26.448, 111.511, -16.946, -84.415, 50.665]
  Set speed (15.0 mm/s)
  Call Extruder(0.015)
  MoveL 594 to (491.4, 508.23, 0.5) mm, rotated rx 0 ry 90 rz 0 deg; joints [-12.94, -26.455, 111.564, -16.919, -84.457, 50.65]
  Set speed (120.0 mm/s)
  MoveL 595 to (491.4, 507.24, 0.5) mm, rotated rx 0 ry 90 rz 0 deg; joints [-12.849, -26.458, 111.59, -16.826, -84.477, 50.636]
  Set speed (15.0 mm/s)
  Call Extruder(0.056)
  MoveL 596 to (492.75, 508.59, 0.5) mm, rotated rx 0 ry 90 rz 0 deg; joints [-12.945, -26.432, 111.395, -16.928, -84.318, 50.693]
  Set speed (120.0 mm/s)
  MoveL 597 to (493.74, 508.59, 0.5) mm, rotated rx 0 ry 90 rz 0 deg; joints [-12.924, -26.415, 111.278, -16.91, -84.221, 50.721]
  Set speed (15.0 mm/s)
  Call Extruder(0.096)
  MoveL 598 to (491.4, 506.25, 0.5) mm, rotated rx 0 ry 90 rz 0 deg; joints [-12.758, -26.462, 111.617, -16.734, -84.497, 50.622]
  Set speed (120.0 mm/s)
  MoveL 599 to (491.4, 505.26, 0.5) mm, rotated rx 0 ry 90 rz 0 deg; joints [-12.666, -26.465, 111.643, -16.641, -84.516, 50.608]
  Set speed (15.0 mm/s)
  Call Extruder(0.137)
  MoveL 600 to (494.73, 508.59, 0.5) mm, rotated rx 0 ry 90 rz 0 deg; joints [-12.903, -26.399, 111.161, -16.892, -84.125, 50.748]
  Set speed (120.0 mm/s)
  MoveL 601 to (495.72, 508.59, 0.5) mm, rotated rx 0 ry 90 rz 0 deg; joints [-12.882, -26.383, 111.044, -16.874, -84.028, 50.776]
  Set speed (15.0 mm/s)
  Call Extruder(0.178)
  MoveL 602 to (491.4, 504.27, 0.5) mm, rotated rx 0 ry 90 rz 0 deg; joints [-12.574, -26.469, 111.669, -16.549, -84.536, 50.594]
  Set speed (120.0 mm/s)
  MoveL 603 to (491.4, 503.28, 0.5) mm, rotated rx 0 ry 90 rz 0 deg; joints [-12.483, -26.472, 111.695, -16.456, -84.555, 50.58]
  Set speed (15.0 mm/s)
  Call Extruder(0.219)
  MoveL 604 to (496.71, 508.59, 0.5) mm, rotated rx 0 ry 90 rz 0 deg; joints [-12.862, -26.366, 110.927, -16.856, -83.931, 50.803]
  Set speed (120.0 mm/s)
  MoveL 605 to (497.7, 508.59, 0.5) mm, rotated rx 0 ry 90 rz 0 deg; joints [-12.841, -26.349, 110.81, -16.838, -83.835, 50.83]
  Set speed (15.0 mm/s)
  Call Extruder(0.259)
  MoveL 606 to (491.4, 502.29, 0.5) mm, rotated rx 0 ry 90 rz 0 deg; joints [-12.391, -26.476, 111.721, -16.364, -84.574, 50.566]
  Set speed (120.0 mm/s)
  MoveL 607 to (491.4, 501.3, 0.5) mm, rotated rx 0 ry 90 rz 0 deg; joints [-12.299, -26.479, 111.746, -16.271, -84.593, 50.553]
  Set speed (15.0 mm/s)
  Call Extruder(0.300)
  MoveL 608 to (498.69, 508.59, 0.5) mm, rotated rx 0 ry 90 rz 0 deg; joints [-12.821, -26.332, 110.693, -16.821, -83.738, 50.858]
  Set speed (120.0 mm/s)
  MoveL 609 to (499.68, 508.59, 0.5) mm, rotated rx 0 ry 90 rz 0 deg; joints [-12.8, -26.315, 110.575, -16.803, -83.642, 50.885]
  Set speed (15.0 mm/s)
  Call Extruder(0.341)
  MoveL 610 to (491.4, 500.31, 0.5) mm, rotated rx 0 ry 90 rz 0 deg; joints [-12.208, -26.483, 111.771, -16.178, -84.612, 50.539]
  Set speed (120.0 mm/s)
  MoveL 611 to (491.4, 499.32, 0.5) mm, rotated rx 0 ry 90 rz 0 deg; joints [-12.116, -26.486, 111.797, -16.085, -84.631, 50.526]
  Set speed (15.0 mm/s)
  Call Extruder(0.382)
  MoveL 612 to (500.67, 508.59, 0.5) mm, rotated rx 0 ry 90 rz 0 deg; joints [-12.78, -26.298, 110.458, -16.786, -83.545, 50.912]
  Set speed (120.0 mm/s)
  MoveL 613 to (501.66, 508.59, 0.5) mm, rotated rx 0 ry 90 rz 0 deg; joints [-12.759, -26.28, 110.34, -16.769, -83.448, 50.939]
  Set speed (15.0 mm/s)
  Call Extruder(0.422)
  MoveL 614 to (491.4, 498.33, 0.5) mm, rotated rx 0 ry 90 rz 0 deg; joints [-12.024, -26.489, 111.821, -15.992, -84.65, 50.513]
  Set speed (120.0 mm/s)
  MoveL 615 to (491.4, 497.34, 0.5) mm, rotated rx 0 ry 90 rz 0 deg; joints [-11.932, -26.493, 111.846, -15.899, -84.668, 50.5]
  Set speed (15.0 mm/s)
  Call Extruder(0.463)
  MoveL 616 to (502.65, 508.59, 0.5) mm, rotated rx 0 ry 90 rz 0 deg; joints [-12.739, -26.262, 110.222, -16.752, -83.352, 50.966]
  Set speed (120.0 mm/s)
  MoveL 617 to (503.64, 508.59, 0.5) mm, rotated rx 0 ry 90 rz 0 deg; joints [-12.719, -26.245, 110.104, -16.735, -83.255, 50.993]
  Set speed (15.0 mm/s)
  Call Extruder(0.504)
  MoveL 618 to (491.4, 496.35, 0.5) mm, rotated rx 0 ry 90 rz 0 deg; joints [-11.839, -26.496, 111.871, -15.806, -84.687, 50.487]
  Set speed (120.0 mm/s)
  MoveL 619 to (491.4, 495.36, 0.5) mm, rotated rx 0 ry 90 rz 0 deg; joints [-11.747, -26.499, 111.895, -15.713, -84.705, 50.474]
  Set speed (15.0 mm/s)
  Call Extruder(0.545)
  MoveL 620 to (504.63, 508.59, 0.5) mm, rotated rx 0 ry 90 rz 0 deg; joints [-12.698, -26.227, 109.986, -16.718, -83.159, 51.02]
  Set speed (120.0 mm/s)
  MoveL 621 to (505.62, 508.59, 0.5) mm, rotated rx 0 ry 90 rz 0 deg; joints [-12.678, -26.208, 109.868, -16.701, -83.062, 51.047]
  Set speed (15.0 mm/s)
  Call Extruder(0.585)
  MoveL 622 to (491.4, 494.37, 0.5) mm, rotated rx 0 ry 90 rz 0 deg; joints [-11.655, -26.502, 111.919, -15.62, -84.723, 50.461]
  Set speed (120.0 mm/s)
  MoveL 623 to (491.4, 493.38, 0.5) mm, rotated rx 0 ry 90 rz 0 deg; joints [-11.563, -26.505, 111.943, -15.527, -84.742, 50.448]
  Set speed (15.0 mm/s)
  Call Extruder(0.626)
  MoveL 624 to (506.61, 508.59, 0.5) mm, rotated rx 0 ry 90 rz 0 deg; joints [-12.658, -26.19, 109.75, -16.684, -82.966, 51.074]
  Set speed (120.0 mm/s)
  MoveL 625 to (507.6, 508.59, 0.5) mm, rotated rx 0 ry 90 rz 0 deg; joints [-12.638, -26.172, 109.631, -16.668, -82.87, 51.1]
  Set speed (15.0 mm/s)
  Call Extruder(0.667)
  MoveL 626 to (491.4, 492.39, 0.5) mm, rotated rx 0 ry 90 rz 0 deg; joints [-11.47, -26.508, 111.967, -15.434, -84.759, 50.436]
  Set speed (120.0 mm/s)
  MoveL 627 to (491.4, 491.4, 0.5) mm, rotated rx 0 ry 90 rz 0 deg; joints [-11.378, -26.512, 111.991, -15.341, -84.777, 50.423]
  Set speed (15.0 mm/s)
  Call Extruder(0.707)
  MoveL 628 to (508.59, 508.59, 0.5) mm, rotated rx 0 ry 90 rz 0 deg; joints [-12.618, -26.153, 109.512, -16.651, -82.773, 51.127]
  Set speed (120.0 mm/s)
